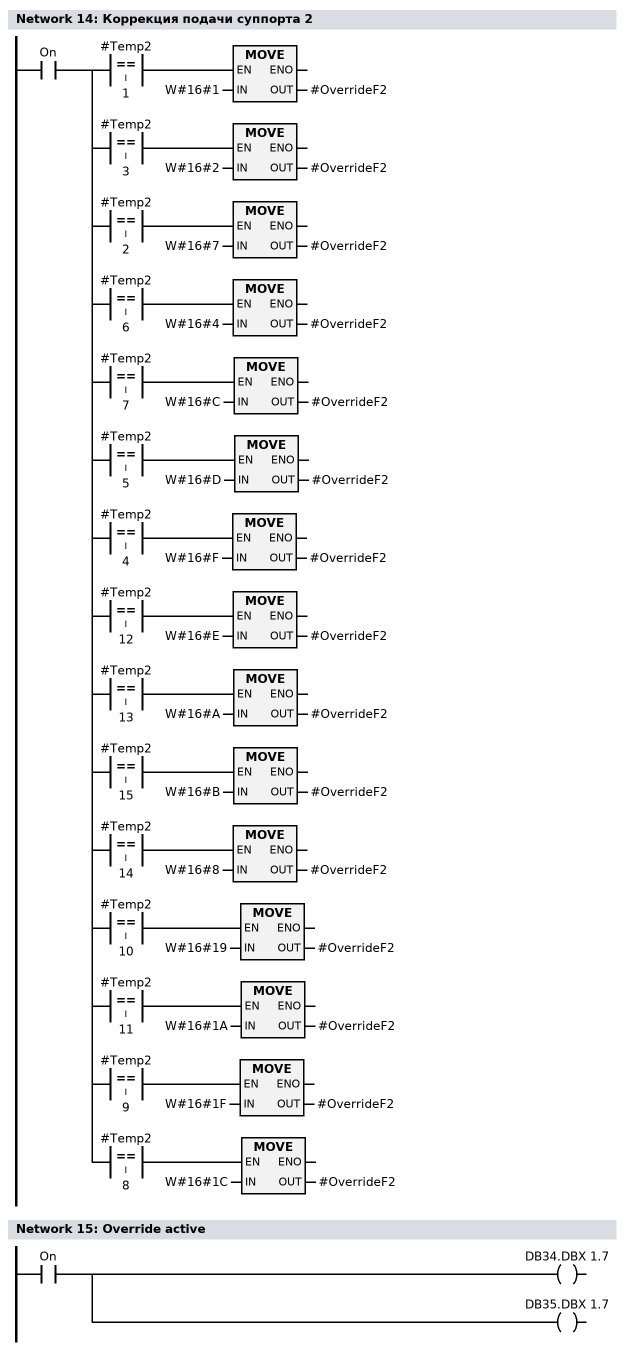
[picture p48: Correction networks 14-15]
NETWORK
TITLE = Коррекция подачи суппорта 2
      A     "On";
      =     L 19.0;
      A     L 19.0;
      A(;
      L     #Temp2;
      L     1;
      ==I;
      );
      JNB   _01b;
      L     W#16#1;
      T     #OverrideF2;
_01b: NOP   0;
      A     L 19.0;
      A(;
      L     #Temp2;
      L     3;
      ==I;
      );
      JNB   _01c;
      L     W#16#2;
      T     #OverrideF2;
_01c: NOP   0;
      A     L 19.0;
      A(;
      L     #Temp2;
      L     2;
      ==I;
      );
      JNB   _01d;
      L     W#16#7;
      T     #OverrideF2;
_01d: NOP   0;
      A     L 19.0;
      A(;
      L     #Temp2;
      L     6;
      ==I;
      );
      JNB   _01e;
      L     W#16#4;
      T     #OverrideF2;
_01e: NOP   0;
      A     L 19.0;
      A(;
      L     #Temp2;
      L     7;
      ==I;
      );
      JNB   _01f;
      L     W#16#C;
      T     #OverrideF2;
_01f: NOP   0;
      A     L 19.0;
      A(;
      L     #Temp2;
      L     5;
      ==I;
      );
      JNB   _020;
      L     W#16#D;
      T     #OverrideF2;
_020: NOP   0;
      A     L 19.0;
      A(;
      L     #Temp2;
      L     4;
      ==I;
      );
      JNB   _021;
      L     W#16#F;
      T     #OverrideF2;
_021: NOP   0;
      A     L 19.0;
      A(;
      L     #Temp2;
      L     12;
      ==I;
      );
      JNB   _022;
      L     W#16#E;
      T     #OverrideF2;
_022: NOP   0;
      A     L 19.0;
      A(;
      L     #Temp2;
      L     13;
      ==I;
      );
      JNB   _023;
      L     W#16#A;
      T     #OverrideF2;
_023: NOP   0;
      A     L 19.0;
      A(;
      L     #Temp2;
      L     15;
      ==I;
      );
      JNB   _024;
      L     W#16#B;
      T     #OverrideF2;
_024: NOP   0;
      A     L 19.0;
      A(;
      L     #Temp2;
      L     14;
      ==I;
      );
      JNB   _025;
      L     W#16#8;
      T     #OverrideF2;
_025: NOP   0;
      A     L 19.0;
      A(;
      L     #Temp2;
      L     10;
      ==I;
      );
      JNB   _026;
      L     W#16#19;
      T     #OverrideF2;
_026: NOP   0;
      A     L 19.0;
      A(;
      L     #Temp2;
      L     11;
      ==I;
      );
      JNB   _027;
      L     W#16#1A;
      T     #OverrideF2;
_027: NOP   0;
      A     L 19.0;
      A(;
      L     #Temp2;
      L     9;
      ==I;
      );
      JNB   _028;
      L     W#16#1F;
      T     #OverrideF2;
_028: NOP   0;
      A     L 19.0;
      A(;
      L     #Temp2;
      L     8;
      ==I;
      );
      JNB   _029;
      L     W#16#1C;
      T     #OverrideF2;
_029: NOP   0;
NETWORK
TITLE = Override active
      A     "On";
      =     DB34.DBX 1.7;
      =     DB35.DBX 1.7;
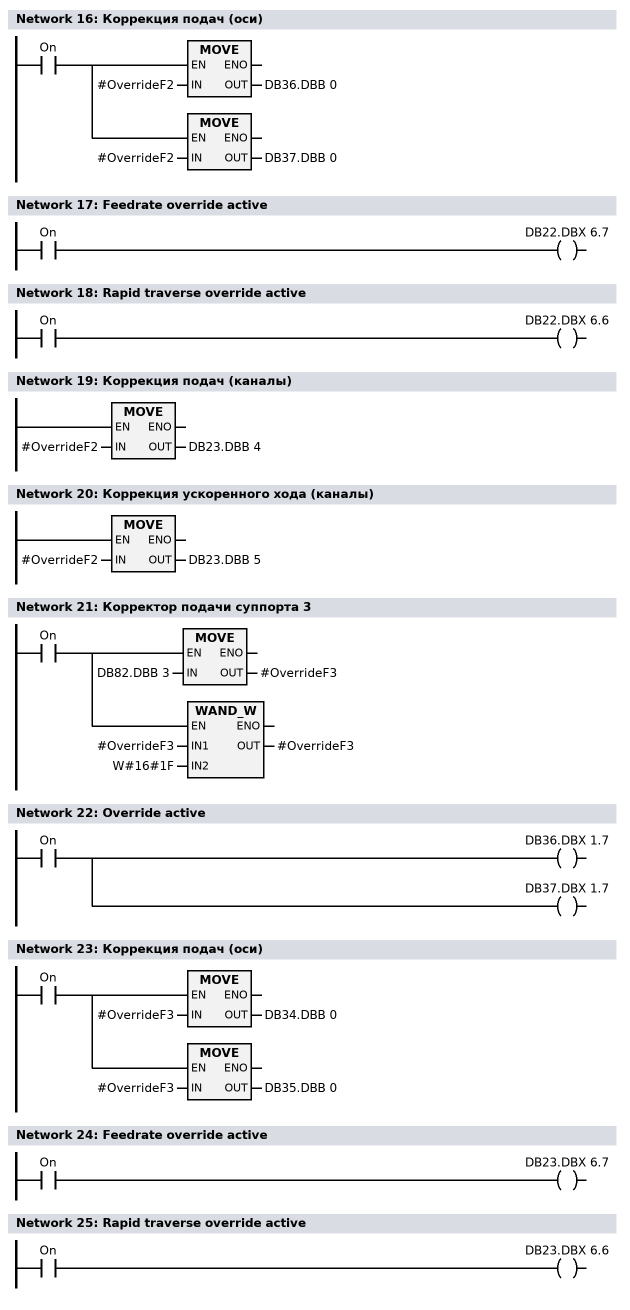
NETWORK
TITLE = Коррекция подач (оси)
      A     "On";
      =     L 19.0;
      A     L 19.0;
      JNB   _02a;
      L     #OverrideF2;
      T     DB36.DBB 0;
_02a: NOP   0;
      A     L 19.0;
      JNB   _02b;
      L     #OverrideF2;
      T     DB37.DBB 0;
_02b: NOP   0;
NETWORK
TITLE = Feedrate override active
      A     "On";
      =     DB22.DBX 6.7;
NETWORK
TITLE = Rapid traverse override active
      A     "On";
      =     DB22.DBX 6.6;
NETWORK
TITLE = Коррекция подач (каналы)
      L     #OverrideF2;
      T     DB23.DBB 4;
      NOP   0;
NETWORK
TITLE = Коррекция ускоренного хода (каналы)
      L     #OverrideF2;
      T     DB23.DBB 5;
      NOP   0;
NETWORK
TITLE = Корректор подачи суппорта 3
      A     "On";
      =     L 19.0;
      A     L 19.0;
      JNB   _02c;
      L     DB82.DBB 3;
      T     #OverrideF3;
_02c: NOP   0;
      A     L 19.0;
      JNB   _02d;
      L     #OverrideF3;
      L     W#16#1F;
      AW;
      T     #OverrideF3;
_02d: NOP   0;
NETWORK
TITLE = Override active
      A     "On";
      =     DB36.DBX 1.7;
      =     DB37.DBX 1.7;
NETWORK
TITLE = Коррекция подач (оси)
      A     "On";
      =     L 19.0;
      A     L 19.0;
      JNB   _02e;
      L     #OverrideF3;
      T     DB34.DBB 0;
_02e: NOP   0;
      A     L 19.0;
      JNB   _02f;
      L     #OverrideF3;
      T     DB35.DBB 0;
_02f: NOP   0;
NETWORK
TITLE = Feedrate override active
      A     "On";
      =     DB23.DBX 6.7;
NETWORK
TITLE = Rapid traverse override active
      A     "On";
      =     DB23.DBX 6.6;
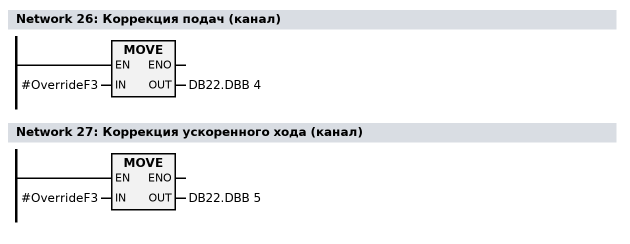
NETWORK
TITLE = Коррекция подач (канал)
      L     #OverrideF3;
      T     DB22.DBB 4;
      NOP   0;
NETWORK
TITLE = Коррекция ускоренного хода (канал)
      L     #OverrideF3;
      T     DB22.DBB 5;
      NOP   0;
NETWORK
TITLE = Корректор подачи суппорта 4
      A     "On";
      =     L 19.0;
      A     L 19.0;
      JNB   _030;
      L     DB82.DBB 0;
      T     #Temp1;
_030: NOP   0;
      A     L 19.0;
      JNB   _031;
      L     #Temp1;
      L     W#16#F0;
      AW;
      T     #Temp1;
_031: NOP   0;
      A     L 19.0;
      JNB   _032;
      L     W#16#4;
      L     #Temp1;
      SRW;
      T     #Temp1;
_032: NOP   0;
      A     L 19.0;
      JNB   _033;
      L     #Temp1;
      T     #Temp2;
_033: NOP   0;
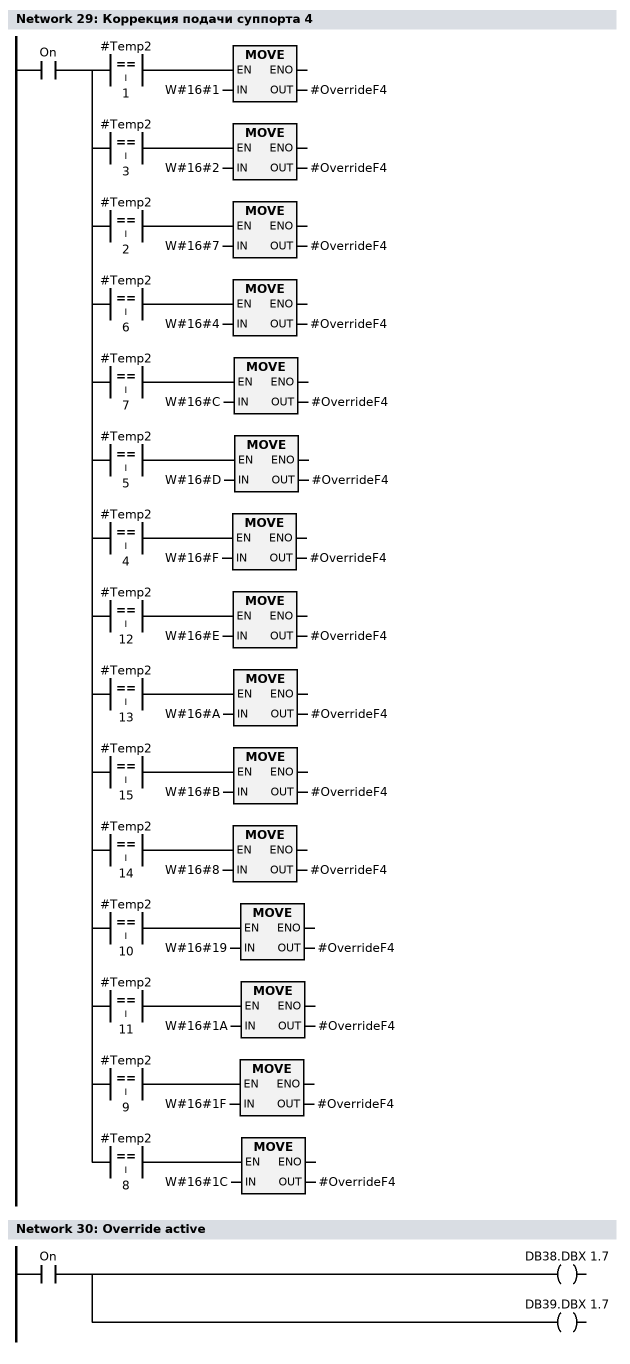
NETWORK
TITLE = Коррекция подачи суппорта 4
      A     "On";
      =     L 19.0;
      A     L 19.0;
      A(;
      L     #Temp2;
      L     1;
      ==I;
      );
      JNB   _034;
      L     W#16#1;
      T     #OverrideF4;
_034: NOP   0;
      A     L 19.0;
      A(;
      L     #Temp2;
      L     3;
      ==I;
      );
      JNB   _035;
      L     W#16#2;
      T     #OverrideF4;
_035: NOP   0;
      A     L 19.0;
      A(;
      L     #Temp2;
      L     2;
      ==I;
      );
      JNB   _036;
      L     W#16#7;
      T     #OverrideF4;
_036: NOP   0;
      A     L 19.0;
      A(;
      L     #Temp2;
      L     6;
      ==I;
      );
      JNB   _037;
      L     W#16#4;
      T     #OverrideF4;
_037: NOP   0;
      A     L 19.0;
      A(;
      L     #Temp2;
      L     7;
      ==I;
      );
      JNB   _038;
      L     W#16#C;
      T     #OverrideF4;
_038: NOP   0;
      A     L 19.0;
      A(;
      L     #Temp2;
      L     5;
      ==I;
      );
      JNB   _039;
      L     W#16#D;
      T     #OverrideF4;
_039: NOP   0;
      A     L 19.0;
      A(;
      L     #Temp2;
      L     4;
      ==I;
      );
      JNB   _03a;
      L     W#16#F;
      T     #OverrideF4;
_03a: NOP   0;
      A     L 19.0;
      A(;
      L     #Temp2;
      L     12;
      ==I;
      );
      JNB   _03b;
      L     W#16#E;
      T     #OverrideF4;
_03b: NOP   0;
      A     L 19.0;
      A(;
      L     #Temp2;
      L     13;
      ==I;
      );
      JNB   _03c;
      L     W#16#A;
      T     #OverrideF4;
_03c: NOP   0;
      A     L 19.0;
      A(;
      L     #Temp2;
      L     15;
      ==I;
      );
      JNB   _03d;
      L     W#16#B;
      T     #OverrideF4;
_03d: NOP   0;
      A     L 19.0;
      A(;
      L     #Temp2;
      L     14;
      ==I;
      );
      JNB   _03e;
      L     W#16#8;
      T     #OverrideF4;
_03e: NOP   0;
      A     L 19.0;
      A(;
      L     #Temp2;
      L     10;
      ==I;
      );
      JNB   _03f;
      L     W#16#19;
      T     #OverrideF4;
_03f: NOP   0;
      A     L 19.0;
      A(;
      L     #Temp2;
      L     11;
      ==I;
      );
      JNB   _040;
      L     W#16#1A;
      T     #OverrideF4;
_040: NOP   0;
      A     L 19.0;
      A(;
      L     #Temp2;
      L     9;
      ==I;
      );
      JNB   _041;
      L     W#16#1F;
      T     #OverrideF4;
_041: NOP   0;
      A     L 19.0;
      A(;
      L     #Temp2;
      L     8;
      ==I;
      );
      JNB   _042;
      L     W#16#1C;
      T     #OverrideF4;
_042: NOP   0;
NETWORK
TITLE = Override active
      A     "On";
      =     DB38.DBX 1.7;
      =     DB39.DBX 1.7;
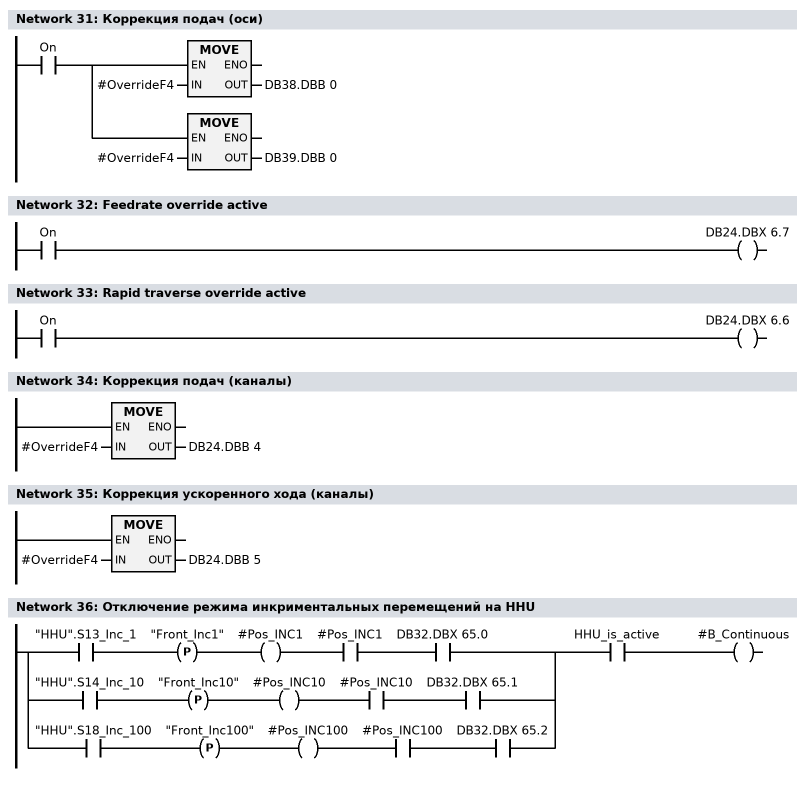
NETWORK
TITLE = Коррекция подач (оси)
      A     "On";
      =     L 19.0;
      A     L 19.0;
      JNB   _043;
      L     #OverrideF4;
      T     DB38.DBB 0;
_043: NOP   0;
      A     L 19.0;
      JNB   _044;
      L     #OverrideF4;
      T     DB39.DBB 0;
_044: NOP   0;
NETWORK
TITLE = Feedrate override active
      A     "On";
      =     DB24.DBX 6.7;
NETWORK
TITLE = Rapid traverse override active
      A     "On";
      =     DB24.DBX 6.6;
NETWORK
TITLE = Коррекция подач (каналы)
      L     #OverrideF4;
      T     DB24.DBB 4;
      NOP   0;
NETWORK
TITLE = Коррекция ускоренного хода (каналы)
      L     #OverrideF4;
      T     DB24.DBB 5;
      NOP   0;
NETWORK
TITLE = Отключение режима инкриментальных перемещений на HHU
      A(;
      A(;
      A     "HHU".S13_Inc_1;
      BLD   100;
      FP    "Front_Inc1";
      );
      =     #Pos_INC1;
      A     #Pos_INC1;
      A     DB32.DBX 65.0;
      O(;
      A(;
      A     "HHU".S14_Inc_10;
      BLD   100;
      FP    "Front_Inc10";
      );
      =     #Pos_INC10;
      A     #Pos_INC10;
      A     DB32.DBX 65.1;
      );
      O(;
      A(;
      A     "HHU".S18_Inc_100;
      BLD   100;
      FP    "Front_Inc100";
      );
      =     #Pos_INC100;
      A     #Pos_INC100;
      A     DB32.DBX 65.2;
      );
      );
      A     "HHU_is_active";
      =     #B_Continuous;
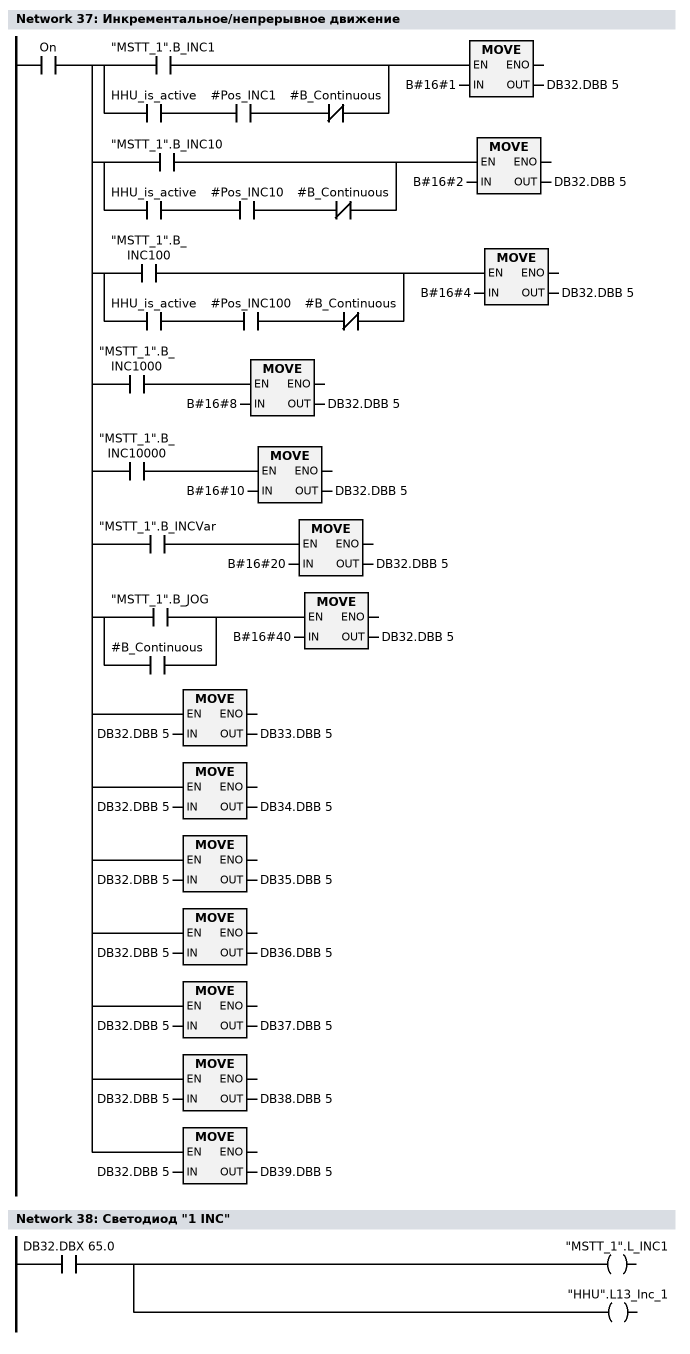
NETWORK
TITLE = Инкрементальное/непрерывное движение
      A     "On";
      =     L 19.0;
      A     L 19.0;
      A(;
      O     "MSTT_1".B_INC1;
      O;
      A     "HHU_is_active";
      A     #Pos_INC1;
      AN    #B_Continuous;
      );
      JNB   _045;
      L     B#16#1;
      T     DB32.DBB 5;
_045: NOP   0;
      A     L 19.0;
      A(;
      O     "MSTT_1".B_INC10;
      O;
      A     "HHU_is_active";
      A     #Pos_INC10;
      AN    #B_Continuous;
      );
      JNB   _046;
      L     B#16#2;
      T     DB32.DBB 5;
_046: NOP   0;
      A     L 19.0;
      A(;
      O     "MSTT_1".B_INC100;
      O;
      A     "HHU_is_active";
      A     #Pos_INC100;
      AN    #B_Continuous;
      );
      JNB   _047;
      L     B#16#4;
      T     DB32.DBB 5;
_047: NOP   0;
      A     L 19.0;
      A     "MSTT_1".B_INC1000;
      JNB   _048;
      L     B#16#8;
      T     DB32.DBB 5;
_048: NOP   0;
      A     L 19.0;
      A     "MSTT_1".B_INC10000;
      JNB   _049;
      L     B#16#10;
      T     DB32.DBB 5;
_049: NOP   0;
      A     L 19.0;
      A     "MSTT_1".B_INCVar;
      JNB   _04a;
      L     B#16#20;
      T     DB32.DBB 5;
_04a: NOP   0;
      A     L 19.0;
      A(;
      O     "MSTT_1".B_JOG;
      O     #B_Continuous;
      );
      JNB   _04b;
      L     B#16#40;
      T     DB32.DBB 5;
_04b: NOP   0;
      A     L 19.0;
      JNB   _04c;
      L     DB32.DBB 5;
      T     DB33.DBB 5;
_04c: NOP   0;
      A     L 19.0;
      JNB   _04d;
      L     DB32.DBB 5;
      T     DB34.DBB 5;
_04d: NOP   0;
      A     L 19.0;
      JNB   _04e;
      L     DB32.DBB 5;
      T     DB35.DBB 5;
_04e: NOP   0;
      A     L 19.0;
      JNB   _04f;
      L     DB32.DBB 5;
      T     DB36.DBB 5;
_04f: NOP   0;
      A     L 19.0;
      JNB   _050;
      L     DB32.DBB 5;
      T     DB37.DBB 5;
_050: NOP   0;
      A     L 19.0;
      JNB   _051;
      L     DB32.DBB 5;
      T     DB38.DBB 5;
_051: NOP   0;
      A     L 19.0;
      JNB   _052;
      L     DB32.DBB 5;
      T     DB39.DBB 5;
_052: NOP   0;
NETWORK
TITLE = Светодиод "1 INC"
      A     DB32.DBX 65.0;
      =     "MSTT_1".L_INC1;
      =     "HHU".L13_Inc_1;
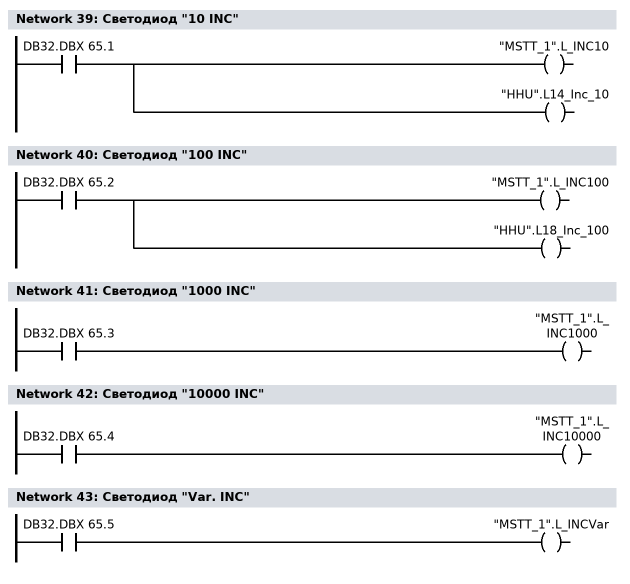
NETWORK
TITLE = Светодиод "10 INC"
      A     DB32.DBX 65.1;
      =     "MSTT_1".L_INC10;
      =     "HHU".L14_Inc_10;
NETWORK
TITLE = Светодиод "100 INC"
      A     DB32.DBX 65.2;
      =     "MSTT_1".L_INC100;
      =     "HHU".L18_Inc_100;
NETWORK
TITLE = Светодиод "1000 INC"
      A     DB32.DBX 65.3;
      =     "MSTT_1".L_INC1000;
NETWORK
TITLE = Светодиод "10000 INC"
      A     DB32.DBX 65.4;
      =     "MSTT_1".L_INC10000;
NETWORK
TITLE = Светодиод "Var. INC"
      A     DB32.DBX 65.5;
      =     "MSTT_1".L_INCVar;
END_FUNCTION

FUNCTION "Others" : VOID	// FC 112
AUTHOR : SEDIN
VERSION : 0.1
VAR_TEMP
  F_Ret_Val : INT ;
  Alarms1 : DINT ;
END_VAR
BEGIN
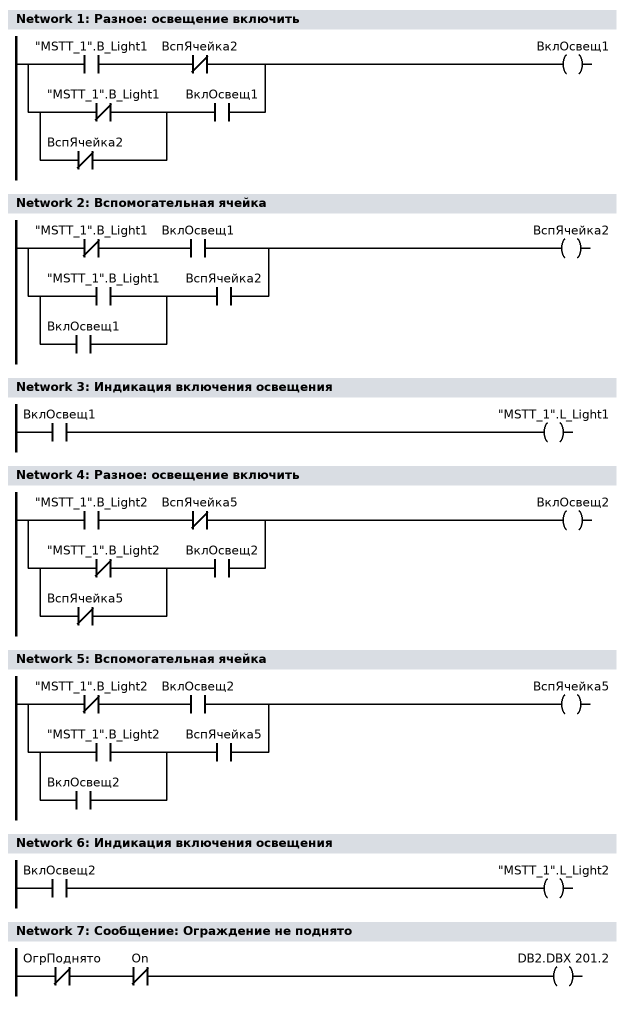
NETWORK
TITLE = Разное: освещение включить
      A     "MSTT_1".B_Light1;
      AN    "ВспЯчейка2";
      O;
      A(;
      ON    "MSTT_1".B_Light1;
      ON    "ВспЯчейка2";
      );
      A     "ВклОсвещ1";
      =     "ВклОсвещ1";
NETWORK
TITLE = Вспомогательная ячейка
      AN    "MSTT_1".B_Light1;
      A     "ВклОсвещ1";
      O;
      A(;
      O     "MSTT_1".B_Light1;
      O     "ВклОсвещ1";
      );
      A     "ВспЯчейка2";
      =     "ВспЯчейка2";
NETWORK
TITLE = Индикация включения освещения
      A     "ВклОсвещ1";
      =     "MSTT_1".L_Light1;
NETWORK
TITLE = Разное: освещение включить
      A     "MSTT_1".B_Light2;
      AN    "ВспЯчейка5";
      O;
      A(;
      ON    "MSTT_1".B_Light2;
      ON    "ВспЯчейка5";
      );
      A     "ВклОсвещ2";
      =     "ВклОсвещ2";
NETWORK
TITLE = Вспомогательная ячейка
      AN    "MSTT_1".B_Light2;
      A     "ВклОсвещ2";
      O;
      A(;
      O     "MSTT_1".B_Light2;
      O     "ВклОсвещ2";
      );
      A     "ВспЯчейка5";
      =     "ВспЯчейка5";
NETWORK
TITLE = Индикация включения освещения
      A     "ВклОсвещ2";
      =     "MSTT_1".L_Light2;
NETWORK
TITLE = Сообщение: Ограждение не поднято
      AN    "ОгрПоднято";
      AN    "On";
      =     DB2.DBX 201.2;
END_FUNCTION

FUNCTION "Hydraullics" : VOID	// FC 115
AUTHOR : SEDIN
VERSION : 0.1
BEGIN
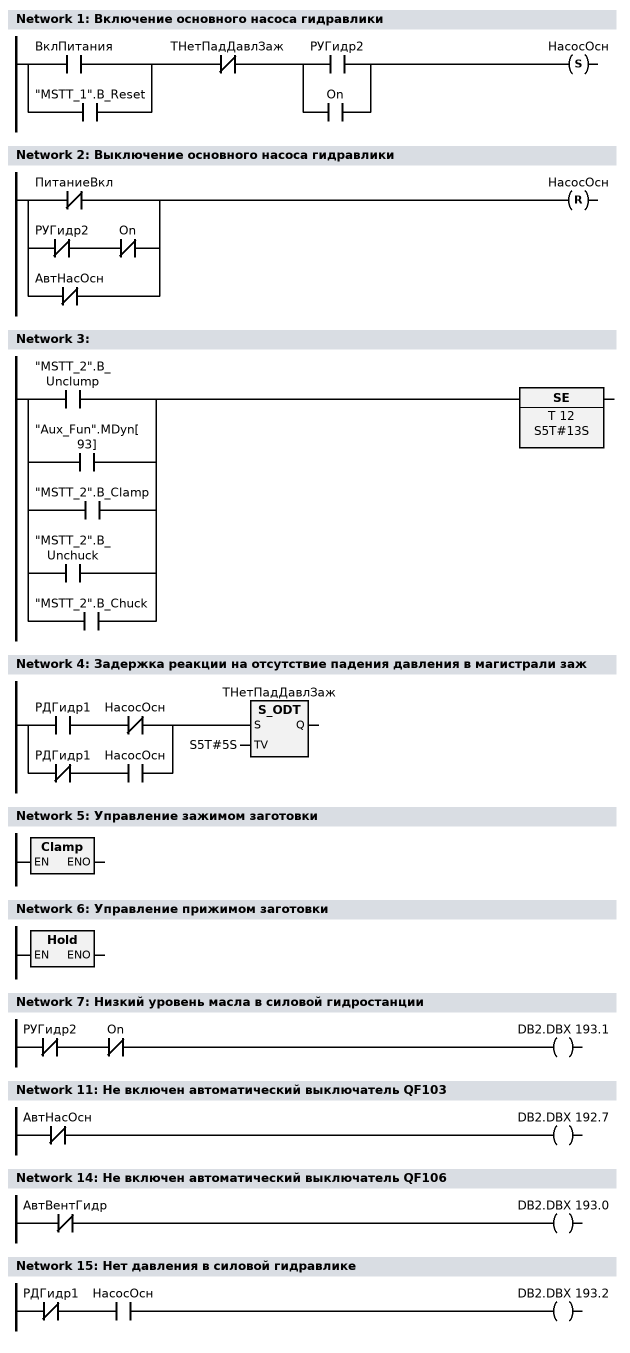
NETWORK
TITLE = Включение основного насоса гидравлики
      A(;
      O     "ВклПитания";
      O     "MSTT_1".B_Reset;
      );
      AN    "ТНетПадДавлЗаж";
      A(;
      O     "РУГидр2";
      O     "On";
      );
      S     "НасосОсн";
NETWORK
TITLE = Выключение основного насоса гидравлики
      ON    "ПитаниеВкл";
      O;
      AN    "РУГидр2";
      AN    "On";
      ON    "АвтНасОсн";
      R     "НасосОсн";
NETWORK
TITLE =
      O     "MSTT_2".B_Unclump;
      O     "Aux_Fun".MDyn[93];
      O     "MSTT_2".B_Clamp;
      O     "MSTT_2".B_Unchuck;
      O     "MSTT_2".B_Chuck;
      L     S5T#13S;
      SE    T 12;
NETWORK
TITLE = Задержка реакции на отсутствие падения давления в магистрали заж
      A(;
      A     "РДГидр1";
      AN    "НасосОсн";
      O;
      AN    "РДГидр1";
      A     "НасосОсн";
      );
      L     S5T#5S;
      SD    "ТНетПадДавлЗаж";
      NOP   0;
      NOP   0;
      NOP   0;
      NOP   0;
NETWORK
TITLE = Управление зажимом заготовки
      CALL  "Clamp";
      NOP   0;
NETWORK
TITLE = Управление прижимом заготовки
      CALL  "Hold";
      NOP   0;
NETWORK
TITLE = Низкий уровень масла в силовой гидростанции
      AN    "РУГидр2";
      AN    "On";
      =     DB2.DBX 193.1;
NETWORK
TITLE = Фильтр SF101 в системе гидравлики засорен
//      AN    "ФильтрSF101"
//      AN    "On"
//      =     "ALMSG_DB".A7001xx[51]
NETWORK
TITLE = Фильтр SF102 в системе гидравлики засорен
//      AN    "ФильтрSF102"
//      AN    "On"
//      =     "ALMSG_DB".A7001xx[52]
NETWORK
TITLE = Фильтр SF103 в системе гидравлики засорен
//      AN    "ФильтрSF103"
//      AN    "On"
//      =     "ALMSG_DB".A7001xx[54]
NETWORK
TITLE = Не включен автоматический выключатель QF103
      AN    "АвтНасОсн";
      =     DB2.DBX 192.7;
NETWORK
TITLE = Не включен автоматический выключатель QF104
//      AN    "АвтНасПод"
//      AN    "On"
//      =     "ALMSG_DB".A7001xx[57]
NETWORK
TITLE = Не включен насос системы гидравлики
//      AN    "НасосОсн"
//      A     "ПитаниеВкл"
//      =     "ALMSG_DB".A7001xx[58]
NETWORK
TITLE = Не включен автоматический выключатель QF106
      AN    "АвтВентГидр";
      =     DB2.DBX 193.0;
NETWORK
TITLE = Нет давления в силовой гидравлике
      AN    "РДГидр1";
      A     "НасосОсн";
      =     DB2.DBX 193.2;
END_FUNCTION

FUNCTION "Clamp" : VOID	// FC 116
AUTHOR : SEDIN
VERSION : 0.1
BEGIN
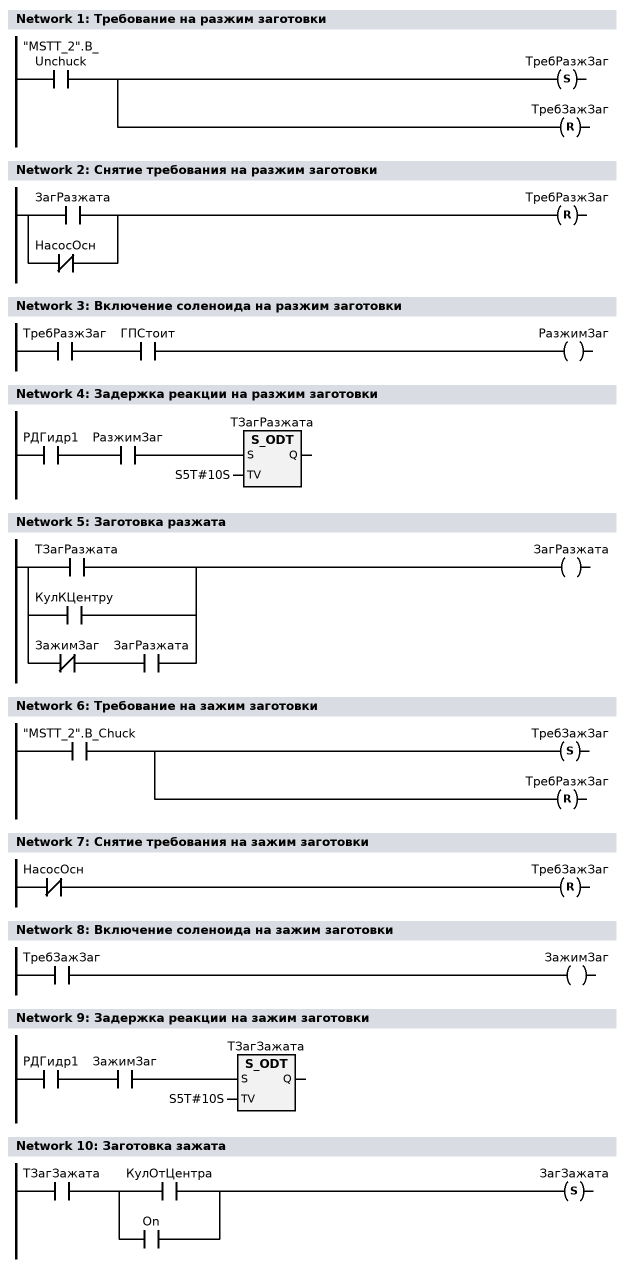
NETWORK
TITLE = Требование на разжим заготовки
      A     "MSTT_2".B_Unchuck;
      S     "ТребРазжЗаг";
      R     "ТребЗажЗаг";
NETWORK
TITLE = Снятие требования на разжим заготовки
      O     "ЗагРазжата";
      ON    "НасосОсн";
      R     "ТребРазжЗаг";
NETWORK
TITLE = Включение соленоида на разжим заготовки
      A     "ТребРазжЗаг";
      A     "ГПСтоит";
      =     "РазжимЗаг";
NETWORK
TITLE = Задержка реакции на разжим заготовки
      A     "РДГидр1";
      A     "РазжимЗаг";
      L     S5T#10S;
      SD    "ТЗагРазжата";
      NOP   0;
      NOP   0;
      NOP   0;
      NOP   0;
NETWORK
TITLE = Заготовка разжата
      O     "ТЗагРазжата";
      O     "КулКЦентру";
      O;
      AN    "ЗажимЗаг";
      A     "ЗагРазжата";
      =     "ЗагРазжата";
NETWORK
TITLE = Требование на зажим заготовки
      A     "MSTT_2".B_Chuck;
      S     "ТребЗажЗаг";
      R     "ТребРазжЗаг";
NETWORK
TITLE = Снятие требования на зажим заготовки
      AN    "НасосОсн";
      R     "ТребЗажЗаг";
NETWORK
TITLE = Включение соленоида на зажим заготовки
      A     "ТребЗажЗаг";
      =     "ЗажимЗаг";
NETWORK
TITLE = Задержка реакции на зажим заготовки
      A     "РДГидр1";
      A     "ЗажимЗаг";
      L     S5T#10S;
      SD    "ТЗагЗажата";
      NOP   0;
      NOP   0;
      NOP   0;
      NOP   0;
NETWORK
TITLE = Заготовка зажата
      A     "ТЗагЗажата";
      A(;
      O     "КулОтЦентра";
      O     "On";
      );
      S     "ЗагЗажата";
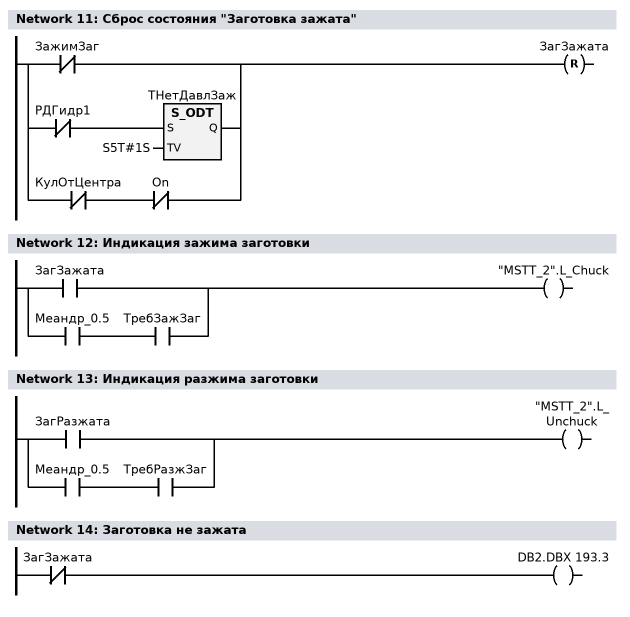
NETWORK
TITLE = Сброс состояния "Заготовка зажата"
      ON    "ЗажимЗаг";
      O(;
      AN    "РДГидр1";
      L     S5T#1S;
      SD    "ТНетДавлЗаж";
      NOP   0;
      NOP   0;
      NOP   0;
      A     "ТНетДавлЗаж";
      );
      O;
      AN    "КулОтЦентра";
      AN    "On";
      R     "ЗагЗажата";
NETWORK
TITLE = Индикация зажима заготовки
      O     "ЗагЗажата";
      O;
      A     "Меандр_0.5";
      A     "ТребЗажЗаг";
      =     "MSTT_2".L_Chuck;
NETWORK
TITLE = Индикация разжима заготовки
      O     "ЗагРазжата";
      O;
      A     "Меандр_0.5";
      A     "ТребРазжЗаг";
      =     "MSTT_2".L_Unchuck;
NETWORK
TITLE = Заготовка не зажата
      AN    "ЗагЗажата";
      =     DB2.DBX 193.3;
END_FUNCTION

FUNCTION "Hold" : VOID	// FC 118
AUTHOR : SEDIN
VERSION : 0.1
BEGIN
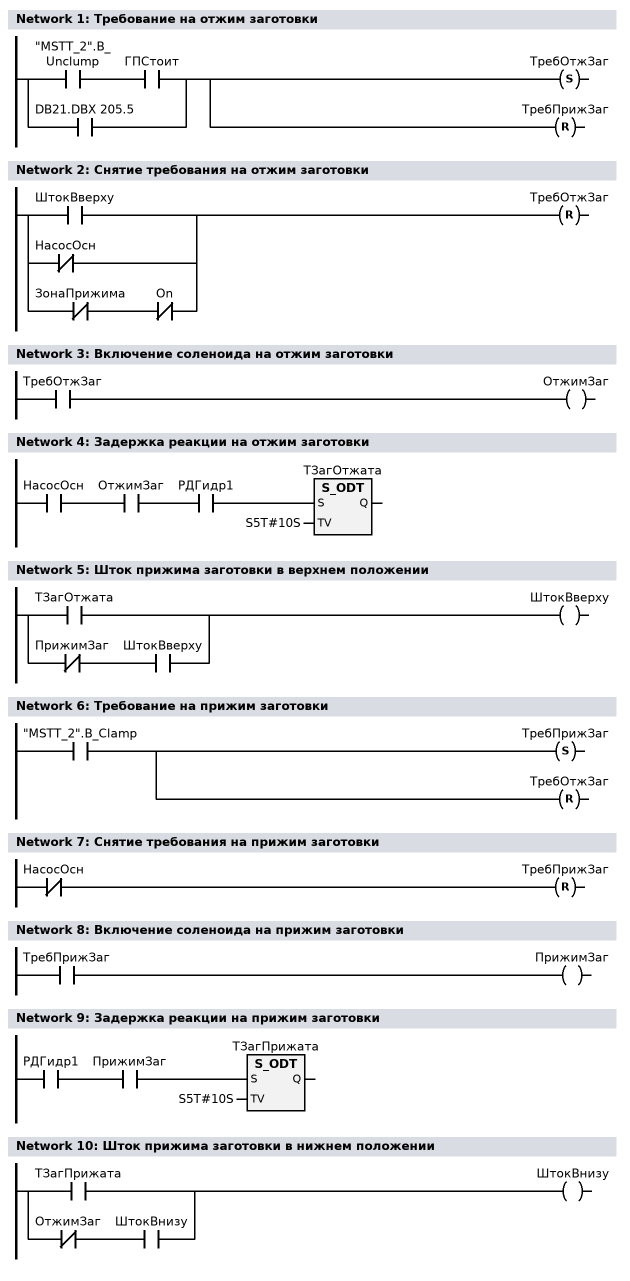
NETWORK
TITLE = Требование на отжим заготовки
      A     "MSTT_2".B_Unclump;
      A     "ГПСтоит";
      O     DB21.DBX 205.5;
      S     "ТребОтжЗаг";
      R     "ТребПрижЗаг";
NETWORK
TITLE = Снятие требования на отжим заготовки
      O     "ШтокВверху";
      ON    "НасосОсн";
      O;
      AN    "ЗонаПрижима";
      AN    "On";
      R     "ТребОтжЗаг";
NETWORK
TITLE = Включение соленоида на отжим заготовки
      A     "ТребОтжЗаг";
      =     "ОтжимЗаг";
NETWORK
TITLE = Задержка реакции на отжим заготовки
      A     "НасосОсн";
      A     "ОтжимЗаг";
      A     "РДГидр1";
      L     S5T#10S;
      SD    "ТЗагОтжата";
      NOP   0;
      NOP   0;
      NOP   0;
      NOP   0;
NETWORK
TITLE = Шток прижима заготовки в верхнем положении
      O     "ТЗагОтжата";
      O;
      AN    "ПрижимЗаг";
      A     "ШтокВверху";
      =     "ШтокВверху";
NETWORK
TITLE = Требование на прижим заготовки
      A     "MSTT_2".B_Clamp;
      S     "ТребПрижЗаг";
      R     "ТребОтжЗаг";
NETWORK
TITLE = Снятие требования на прижим заготовки
      AN    "НасосОсн";
      R     "ТребПрижЗаг";
NETWORK
TITLE = Включение соленоида на прижим заготовки
      A     "ТребПрижЗаг";
      =     "ПрижимЗаг";
NETWORK
TITLE = Задержка реакции на прижим заготовки
      A     "РДГидр1";
      A     "ПрижимЗаг";
      L     S5T#10S;
      SD    "ТЗагПрижата";
      NOP   0;
      NOP   0;
      NOP   0;
      NOP   0;
NETWORK
TITLE = Шток прижима заготовки в нижнем положении
      O     "ТЗагПрижата";
      O;
      AN    "ОтжимЗаг";
      A     "ШтокВнизу";
      =     "ШтокВнизу";
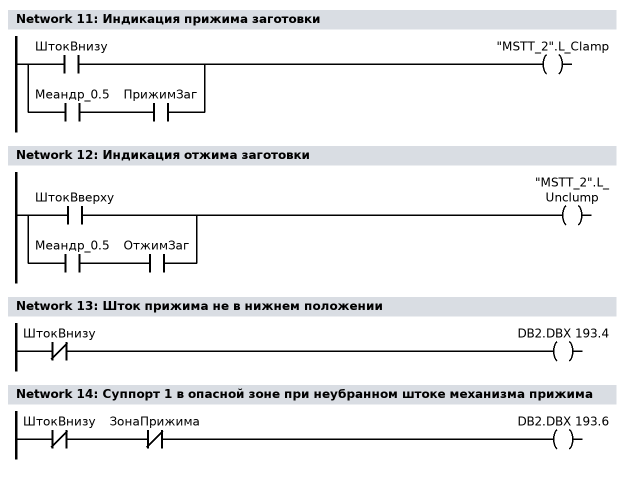
NETWORK
TITLE = Индикация прижима заготовки
      O     "ШтокВнизу";
      O;
      A     "Меандр_0.5";
      A     "ПрижимЗаг";
      =     "MSTT_2".L_Clamp;
NETWORK
TITLE = Индикация отжима заготовки
      O     "ШтокВверху";
      O;
      A     "Меандр_0.5";
      A     "ОтжимЗаг";
      =     "MSTT_2".L_Unclump;
NETWORK
TITLE = Шток прижима не в нижнем положении
      AN    "ШтокВнизу";
      =     DB2.DBX 193.4;
NETWORK
TITLE = Суппорт 1 в опасной зоне при неубранном штоке механизма прижима
      AN    "ШтокВнизу";
      AN    "ЗонаПрижима";
      =     DB2.DBX 193.6;
END_FUNCTION

FUNCTION "Table_Lub" : VOID	// FC 120
AUTHOR : SEDIN
VERSION : 0.1
BEGIN
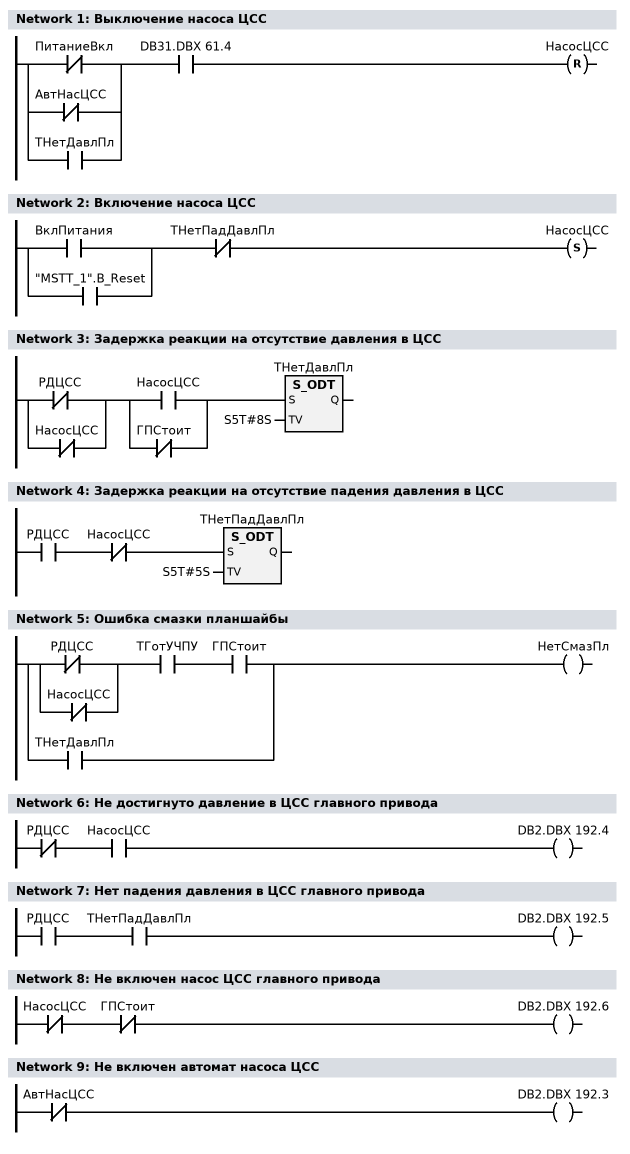
NETWORK
TITLE = Выключение насоса ЦСС
      A(;
      ON    "ПитаниеВкл";
      ON    "АвтНасЦСС";
      O     "ТНетДавлПл";
      );
      A     DB31.DBX 61.4;
      R     "НасосЦСС";
NETWORK
TITLE = Включение насоса ЦСС
      A(;
      O     "ВклПитания";
      O     "MSTT_1".B_Reset;
      );
      AN    "ТНетПадДавлПл";
      S     "НасосЦСС";
NETWORK
TITLE = Задержка реакции на отсутствие давления в ЦСС
      A(;
      ON    "РДЦСС";
      ON    "НасосЦСС";
      );
      A(;
      O     "НасосЦСС";
      ON    "ГПСтоит";
      );
      L     S5T#8S;
      SD    "ТНетДавлПл";
      NOP   0;
      NOP   0;
      NOP   0;
      NOP   0;
NETWORK
TITLE = Задержка реакции на отсутствие падения давления в ЦСС
      A     "РДЦСС";
      AN    "НасосЦСС";
      L     S5T#5S;
      SD    "ТНетПадДавлПл";
      NOP   0;
      NOP   0;
      NOP   0;
      NOP   0;
NETWORK
TITLE = Ошибка смазки планшайбы
      A(;
      ON    "РДЦСС";
      ON    "НасосЦСС";
      );
      A     "ТГотУЧПУ";
      A     "ГПСтоит";
      O     "ТНетДавлПл";
      =     "НетСмазПл";
NETWORK
TITLE = Не достигнуто давление в ЦСС главного привода
      AN    "РДЦСС";
      A     "НасосЦСС";
      =     DB2.DBX 192.4;
NETWORK
TITLE = Нет падения давления в ЦСС главного привода
      A     "РДЦСС";
      A     "ТНетПадДавлПл";
      =     DB2.DBX 192.5;
NETWORK
TITLE = Не включен насос ЦСС главного привода
      AN    "НасосЦСС";
      AN    "ГПСтоит";
      =     DB2.DBX 192.6;
NETWORK
TITLE = Не включен автомат насоса ЦСС
      AN    "АвтНасЦСС";
      =     DB2.DBX 192.3;
END_FUNCTION

FUNCTION "MiniHHU" : VOID	// FC 121
VERSION : 0.1
BEGIN
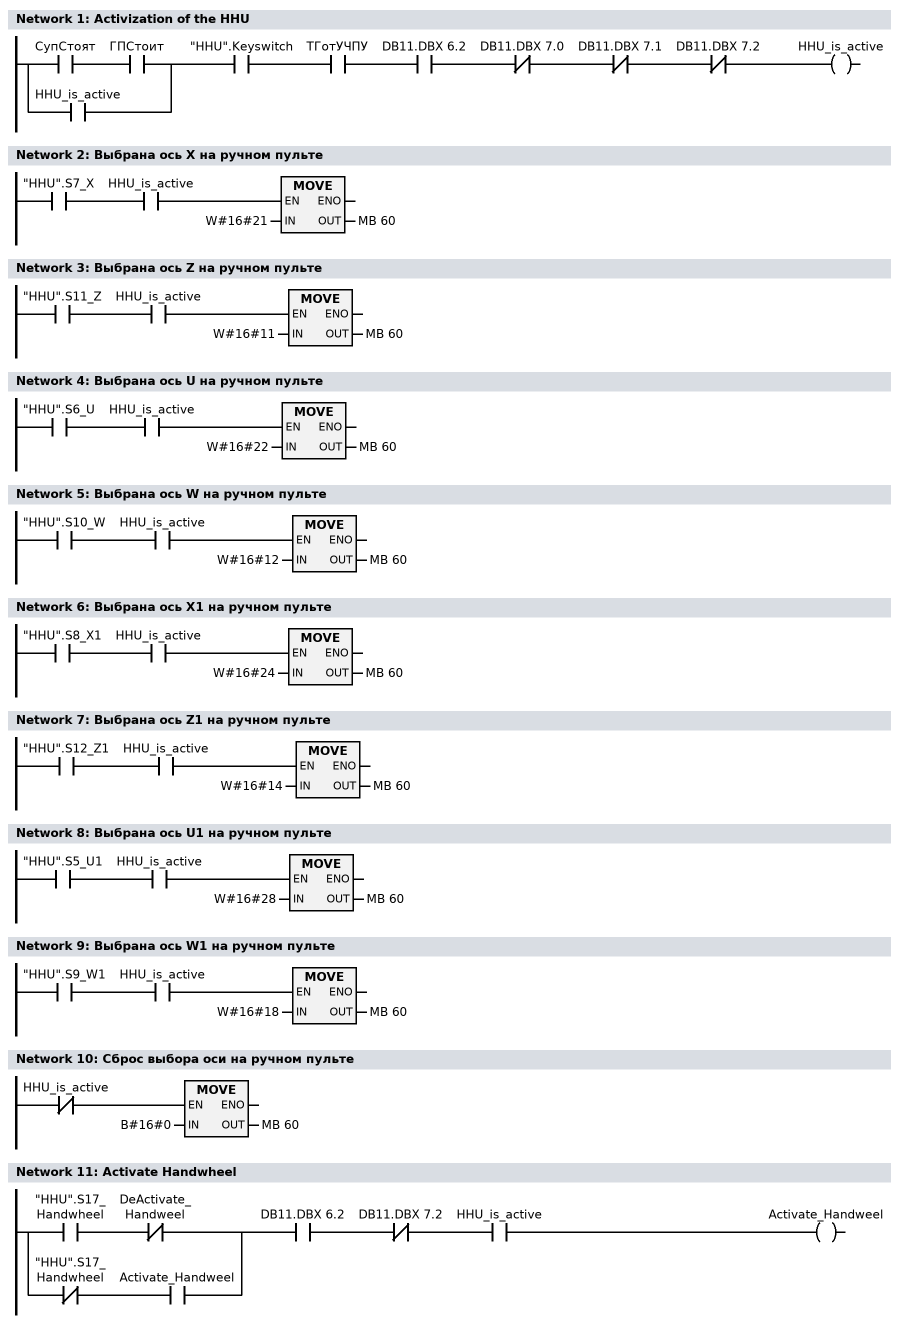
NETWORK
TITLE = Activization of the HHU
      A(;
      A     "СупСтоят";
      A     "ГПСтоит";
      O     "HHU_is_active";
      );
      A     "HHU".Keyswitch;
      A     "ТГотУЧПУ";
      A     DB11.DBX 6.2;
      AN    DB11.DBX 7.0;
      AN    DB11.DBX 7.1;
      AN    DB11.DBX 7.2;
      =     "HHU_is_active";
NETWORK
TITLE = Выбрана ось X на ручном пульте
      A     "HHU".S7_X;
      A     "HHU_is_active";
      JNB   _001;
      L     W#16#21;
      T     MB 60;
_001: NOP   0;
NETWORK
TITLE = Выбрана ось Z на ручном пульте
      A     "HHU".S11_Z;
      A     "HHU_is_active";
      JNB   _002;
      L     W#16#11;
      T     MB 60;
_002: NOP   0;
NETWORK
TITLE = Выбрана ось U на ручном пульте
      A     "HHU".S6_U;
      A     "HHU_is_active";
      JNB   _003;
      L     W#16#22;
      T     MB 60;
_003: NOP   0;
NETWORK
TITLE = Выбрана ось W на ручном пульте
      A     "HHU".S10_W;
      A     "HHU_is_active";
      JNB   _004;
      L     W#16#12;
      T     MB 60;
_004: NOP   0;
NETWORK
TITLE = Выбрана ось X1 на ручном пульте
      A     "HHU".S8_X1;
      A     "HHU_is_active";
      JNB   _005;
      L     W#16#24;
      T     MB 60;
_005: NOP   0;
NETWORK
TITLE = Выбрана ось Z1 на ручном пульте
      A     "HHU".S12_Z1;
      A     "HHU_is_active";
      JNB   _006;
      L     W#16#14;
      T     MB 60;
_006: NOP   0;
NETWORK
TITLE = Выбрана ось U1 на ручном пульте
      A     "HHU".S5_U1;
      A     "HHU_is_active";
      JNB   _007;
      L     W#16#28;
      T     MB 60;
_007: NOP   0;
NETWORK
TITLE = Выбрана ось W1 на ручном пульте
      A     "HHU".S9_W1;
      A     "HHU_is_active";
      JNB   _008;
      L     W#16#18;
      T     MB 60;
_008: NOP   0;
NETWORK
TITLE = Сброс выбора оси на ручном пульте
      AN    "HHU_is_active";
      JNB   _009;
      L     B#16#0;
      T     MB 60;
_009: NOP   0;
NETWORK
TITLE = Activate Handwheel
      A(;
      A     "HHU".S17_Handwheel;
      AN    "DeActivate_Handweel";
      O;
      AN    "HHU".S17_Handwheel;
      A     "Activate_Handweel";
      );
      A     DB11.DBX 6.2;
      AN    DB11.DBX 7.2;
      A     "HHU_is_active";
      =     "Activate_Handweel";
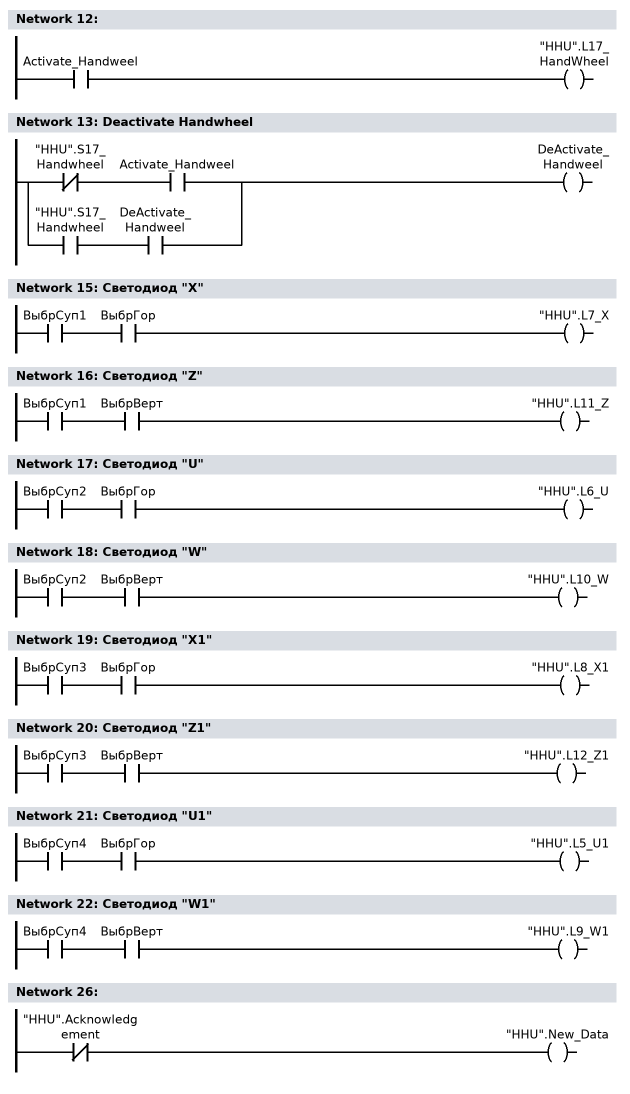
NETWORK
TITLE =
      A     "Activate_Handweel";
      =     "HHU".L17_HandWheel;
NETWORK
TITLE = Deactivate Handwheel
      AN    "HHU".S17_Handwheel;
      A     "Activate_Handweel";
      O;
      A     "HHU".S17_Handwheel;
      A     "DeActivate_Handweel";
      =     "DeActivate_Handweel";
NETWORK
TITLE =
NETWORK
TITLE = Светодиод "X"
      A     "ВыбрСуп1";
      A     "ВыбрГор";
      =     "HHU".L7_X;
NETWORK
TITLE = Светодиод "Z"
      A     "ВыбрСуп1";
      A     "ВыбрВерт";
      =     "HHU".L11_Z;
NETWORK
TITLE = Светодиод "U"
      A     "ВыбрСуп2";
      A     "ВыбрГор";
      =     "HHU".L6_U;
NETWORK
TITLE = Светодиод "W"
      A     "ВыбрСуп2";
      A     "ВыбрВерт";
      =     "HHU".L10_W;
NETWORK
TITLE = Светодиод "X1"
      A     "ВыбрСуп3";
      A     "ВыбрГор";
      =     "HHU".L8_X1;
NETWORK
TITLE = Светодиод "Z1"
      A     "ВыбрСуп3";
      A     "ВыбрВерт";
      =     "HHU".L12_Z1;
NETWORK
TITLE = Светодиод "U1"
      A     "ВыбрСуп4";
      A     "ВыбрГор";
      =     "HHU".L5_U1;
NETWORK
TITLE = Светодиод "W1"
      A     "ВыбрСуп4";
      A     "ВыбрВерт";
      =     "HHU".L9_W1;
NETWORK
TITLE =
      SET;
      S     DB83.DBX 6.7;
      A     "HHU".Acknowledgement;
      FP    "HHU".Auxilary[1];
      =     L 14.0;
      A     L 14.0;
      BLD   102;
      R     "HHU".New_Data;
      A     L 14.0;
      JNB   _010;
      L     DB83.DBB 7;
      INC   1;
      T     DB83.DBB 7;
_010: NOP   0;
      A     L 14.0;
      A     "HHU".Reserved_7_2;
      R     "HHU".Reserved_7_2;
NETWORK
TITLE =
      AN    "HHU".Keyswitch;
      =     L 15.0;
      A     L 15.0;
      AN    "HHU".Selection_Line_1_2;
      AN    "HHU".Selection_Line_3_4;
      JNB   _012;
      L     '$00';
      T     "HHU".DataLine[1];
      T     "HHU".DataLine[2];
      T     "HHU".DataLine[3];
      T     "HHU".DataLine[4];
      T     "HHU".DataLine[5];
      T     "HHU".DataLine[6];
      T     "HHU".DataLine[7];
      T     "HHU".DataLine[8];
      T     "HHU".DataLine[9];
      T     "HHU".DataLine[10];
      T     "HHU".DataLine[11];
      T     "HHU".DataLine[12];
      T     "HHU".DataLine[13];
      T     "HHU".DataLine[14];
      T     "HHU".DataLine[15];
      T     "HHU".DataLine[16];
_012: NOP   0;
      A     L 15.0;
      A     "HHU".Selection_Line_1_2;
      AN    "HHU".Selection_Line_3_4;
      JNB   _013;
      L     '$00';
      T     "HHU".DataLine[1];
      T     "HHU".DataLine[2];
      T     "HHU".DataLine[3];
      L     't';
      T     "HHU".DataLine[4];
      L     'o';
      T     "HHU".DataLine[5];
      L     'n';
      T     "HHU".DataLine[6];
      L     '$00';
      T     "HHU".DataLine[7];
      L     's';
      T     "HHU".DataLine[8];
      L     'i';
      T     "HHU".DataLine[9];
      L     '$00';
      T     "HHU".DataLine[10];
      L     '2';
      T     "HHU".DataLine[11];
      L     'T';
      T     "HHU".DataLine[12];
      L     'H';
      T     "HHU".DataLine[13];
      L     '$00';
      T     "HHU".DataLine[14];
      T     "HHU".DataLine[15];
      T     "HHU".DataLine[16];
_013: NOP   0;
      A     L 15.0;
      AN    "HHU".Selection_Line_1_2;
      A     "HHU".Selection_Line_3_4;
      JNB   _014;
      L     '$00';
      T     "HHU".DataLine[1];
      T     "HHU".DataLine[2];
      T     "HHU".DataLine[3];
      T     "HHU".DataLine[4];
      T     "HHU".DataLine[5];
      L     'e';
      T     "HHU".DataLine[6];
      L     'v';
      T     "HHU".DataLine[7];
      L     'i';
      T     "HHU".DataLine[8];
      L     't';
      T     "HHU".DataLine[9];
      L     'c';
      T     "HHU".DataLine[10];
      L     'a';
      T     "HHU".DataLine[11];
      L     '$00';
      T     "HHU".DataLine[12];
      T     "HHU".DataLine[13];
      T     "HHU".DataLine[14];
      T     "HHU".DataLine[15];
      T     "HHU".DataLine[16];
_014: NOP   0;
      A     L 15.0;
      A     "HHU".Selection_Line_1_2;
      A     "HHU".Selection_Line_3_4;
      JNB   _015;
      L     '$00';
      T     "HHU".DataLine[1];
      T     "HHU".DataLine[2];
      T     "HHU".DataLine[3];
      T     "HHU".DataLine[4];
      T     "HHU".DataLine[5];
      T     "HHU".DataLine[6];
      T     "HHU".DataLine[7];
      T     "HHU".DataLine[8];
      T     "HHU".DataLine[9];
      T     "HHU".DataLine[10];
      T     "HHU".DataLine[11];
      T     "HHU".DataLine[12];
      T     "HHU".DataLine[13];
      T     "HHU".DataLine[14];
      T     "HHU".DataLine[15];
      T     "HHU".DataLine[16];
_015: NOP   0;
NETWORK
TITLE =
      A     "HHU".Keyswitch;
      =     L 15.0;
      A     L 15.0;
      AN    "HHU".Selection_Line_1_2;
      AN    "HHU".Selection_Line_3_4;
      JNB   _016;
      L     '$00';
      T     "HHU".DataLine[1];
      T     "HHU".DataLine[2];
      T     "HHU".DataLine[3];
      T     "HHU".DataLine[4];
      T     "HHU".DataLine[5];
      T     "HHU".DataLine[6];
      T     "HHU".DataLine[7];
      T     "HHU".DataLine[8];
      T     "HHU".DataLine[9];
      T     "HHU".DataLine[10];
      T     "HHU".DataLine[11];
      T     "HHU".DataLine[12];
      T     "HHU".DataLine[13];
      T     "HHU".DataLine[14];
      T     "HHU".DataLine[15];
      T     "HHU".DataLine[16];
_016: NOP   0;
      A     L 15.0;
      A     "HHU".Selection_Line_1_2;
      AN    "HHU".Selection_Line_3_4;
      JNB   _017;
      L     '$00';
      T     "HHU".DataLine[1];
      T     "HHU".DataLine[2];
      T     "HHU".DataLine[3];
      T     "HHU".DataLine[4];
      T     "HHU".DataLine[5];
      L     's';
      T     "HHU".DataLine[6];
      L     'i';
      T     "HHU".DataLine[7];
      L     '$00';
      T     "HHU".DataLine[8];
      L     '2';
      T     "HHU".DataLine[9];
      L     'T';
      T     "HHU".DataLine[10];
      L     'H';
      T     "HHU".DataLine[11];
      L     '$00';
      T     "HHU".DataLine[12];
      T     "HHU".DataLine[13];
      T     "HHU".DataLine[14];
      T     "HHU".DataLine[15];
      T     "HHU".DataLine[16];
_017: NOP   0;
      A     L 15.0;
      AN    "HHU".Selection_Line_1_2;
      A     "HHU".Selection_Line_3_4;
      JNB   _018;
      L     '$00';
      T     "HHU".DataLine[1];
      T     "HHU".DataLine[2];
      T     "HHU".DataLine[3];
      T     "HHU".DataLine[4];
      T     "HHU".DataLine[5];
      L     'e';
      T     "HHU".DataLine[6];
      L     'v';
      T     "HHU".DataLine[7];
      L     'i';
      T     "HHU".DataLine[8];
      L     't';
      T     "HHU".DataLine[9];
      L     'c';
      T     "HHU".DataLine[10];
      L     'a';
      T     "HHU".DataLine[11];
      L     '$00';
      T     "HHU".DataLine[12];
      T     "HHU".DataLine[13];
      T     "HHU".DataLine[14];
      T     "HHU".DataLine[15];
      T     "HHU".DataLine[16];
_018: NOP   0;
      A     L 15.0;
      A     "HHU".Selection_Line_1_2;
      A     "HHU".Selection_Line_3_4;
      JNB   _019;
      L     '$00';
      T     "HHU".DataLine[1];
      T     "HHU".DataLine[2];
      T     "HHU".DataLine[3];
      T     "HHU".DataLine[4];
      T     "HHU".DataLine[5];
      T     "HHU".DataLine[6];
      T     "HHU".DataLine[7];
      T     "HHU".DataLine[8];
      T     "HHU".DataLine[9];
      T     "HHU".DataLine[10];
      T     "HHU".DataLine[11];
      T     "HHU".DataLine[12];
      T     "HHU".DataLine[13];
      T     "HHU".DataLine[14];
      T     "HHU".DataLine[15];
      T     "HHU".DataLine[16];
_019: NOP   0;
NETWORK
TITLE =
      AN    "HHU".Acknowledgement;
      =     "HHU".New_Data;
NETWORK
TITLE =
NETWORK
TITLE =
NETWORK
TITLE =
NETWORK
TITLE =
NETWORK
TITLE =
NETWORK
TITLE =
NETWORK
TITLE =
NETWORK
TITLE =
NETWORK
TITLE =
NETWORK
TITLE =
NETWORK
TITLE =
END_FUNCTION

FUNCTION "Share_Ctrll" : VOID	// FC 150
VERSION : 0.1
VAR_TEMP
  Ret_SFC1 : INT ;
  CDT_SFC1 : DATE_AND_TIME ;
  Ret_SFC20 : INT ;
  Ret_1 : WORD ;	//Результат работы блока FB2
  Temp1 : REAL ;
  ErrWrite : BOOL ;
  ERRCODE : INT ;
END_VAR
BEGIN
NETWORK
TITLE =
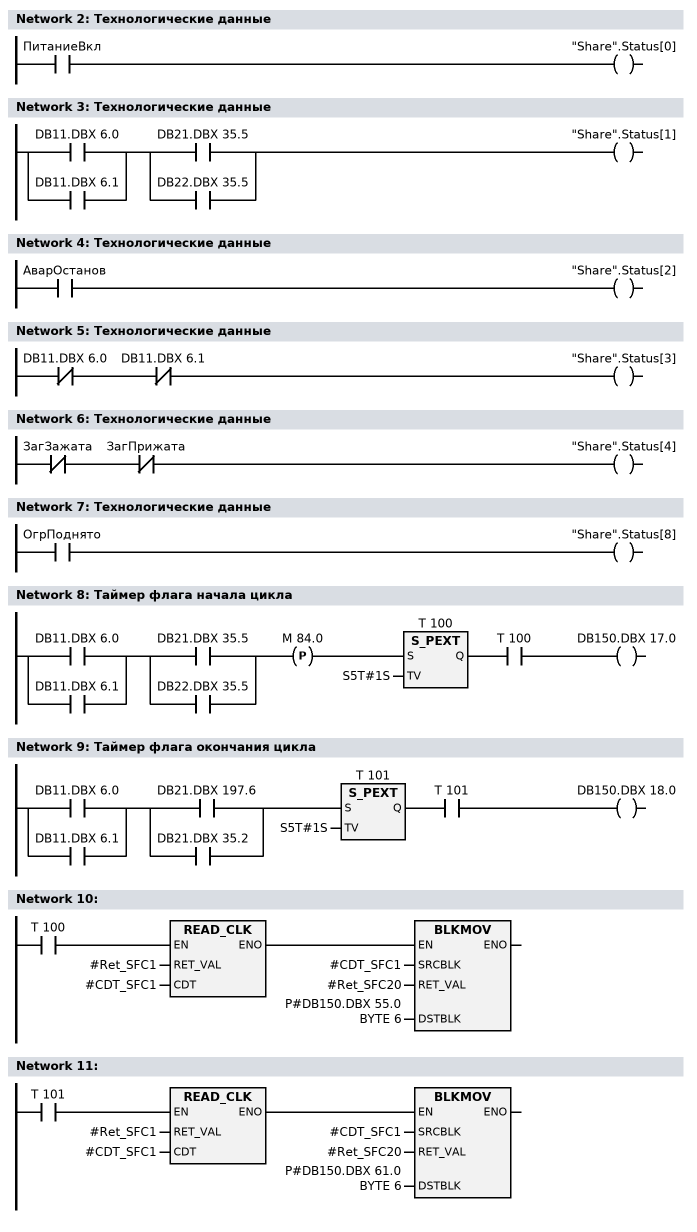
NETWORK
TITLE = Технологические данные
      A     "ПитаниеВкл";
      =     "Share".Status[0];
NETWORK
TITLE = Технологические данные
      A(;
      O     DB11.DBX 6.0;
      O     DB11.DBX 6.1;
      );
      A(;
      O     DB21.DBX 35.5;
      O     DB22.DBX 35.5;
      );
      =     "Share".Status[1];
NETWORK
TITLE = Технологические данные
//Авария.
      A     "АварОстанов";
      =     "Share".Status[2];
NETWORK
TITLE = Технологические данные
//Станок не в автомате. 
      AN    DB11.DBX 6.0;
      AN    DB11.DBX 6.1;
      =     "Share".Status[3];
NETWORK
TITLE = Технологические данные
//Заготовка не зажата.
      AN    "ЗагЗажата";
      AN    "ЗагПрижата";
      =     "Share".Status[4];
NETWORK
TITLE = Технологические данные
//Ограждение закрыто.
      A     "ОгрПоднято";
      =     "Share".Status[8];
NETWORK
TITLE = Таймер флага начала цикла
      A(;
      A(;
      O     DB11.DBX 6.0;
      O     DB11.DBX 6.1;
      );
      A(;
      O     DB21.DBX 35.5;
      O     DB22.DBX 35.5;
      );
      FP    M 84.0;
      L     S5T#1S;
      SE    T 100;
      NOP   0;
      NOP   0;
      NOP   0;
      A     T 100;
      );
      A     T 100;
      =     DB150.DBX 17.0;
NETWORK
TITLE = Таймер флага окончания цикла
      A(;
      A(;
      O     DB11.DBX 6.0;
      O     DB11.DBX 6.1;
      );
      A(;
      O     DB21.DBX 197.6;
      O     DB21.DBX 35.2;
      );
      L     S5T#1S;
      SE    T 101;
      NOP   0;
      NOP   0;
      NOP   0;
      A     T 101;
      );
      A     T 101;
      =     DB150.DBX 18.0;
NETWORK
TITLE =
      A(;
      A     T 100;
      JNB   _001;
      CALL  "READ_CLK" (
           RET_VAL                  := #Ret_SFC1,
           CDT                      := #CDT_SFC1);
_001: A     BR;
      );
      JNB   _002;
      CALL  "BLKMOV" (
           SRCBLK                   := #CDT_SFC1,
           RET_VAL                  := #Ret_SFC20,
           DSTBLK                   := P#DB150.DBX 55.0 BYTE 6);
_002: NOP   0;
NETWORK
TITLE =
      A(;
      A     T 101;
      JNB   _003;
      CALL  "READ_CLK" (
           RET_VAL                  := #Ret_SFC1,
           CDT                      := #CDT_SFC1);
_003: A     BR;
      );
      JNB   _004;
      CALL  "BLKMOV" (
           SRCBLK                   := #CDT_SFC1,
           RET_VAL                  := #Ret_SFC20,
           DSTBLK                   := P#DB150.DBX 61.0 BYTE 6);
_004: NOP   0;
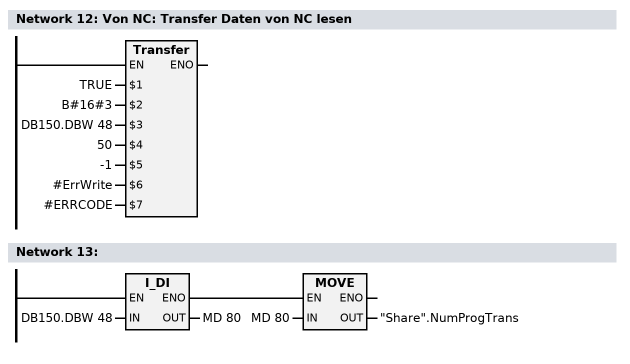
NETWORK
TITLE = Von NC: Transfer Daten von NC lesen
//$A_DBW50: Идентификатор программы обработки
      CALL  "Transfer" (
           $1                       := TRUE,
           $2                       := B#16#3,
           $3                       := DB150.DBW 48,
           $4                       := 50,
           $5                       := -1,
           $6                       := #ErrWrite,
           $7                       := #ERRCODE);
      NOP   0;
NETWORK
TITLE =
//Преобразование идентификатора программы обработки из Integer в DInteger
//
      A(;
      L     DB150.DBW 48;
      ITD;
      T     MD 80;
      SET;
      SAVE;
      CLR;
      A     BR;
      );
      JNB   _005;
      L     MD 80;
      T     "Share".NumProgTrans;
_005: NOP   0;
END_FUNCTION

// FC 1005: know-how protected block, not included

// FC 1006: know-how protected block, not included

// FC 1007: know-how protected block, not included

// FC 1008: know-how protected block, not included

// FC 1010: know-how protected block, not included

DATA_BLOCK DB 4
AUTHOR : NUMERIK
FAMILY : _800D
NAME : Basics
VERSION : 2.7
  STRUCT
   BOfeld0 : WORD  := W#16#CD54;	//Channel 1-8 ever 18 Bits
   BOfeld2 : WORD  := W#16#3553;
   BOfeld4 : WORD  := W#16#D54C;
   BOfeld6 : WORD  := W#16#5533;
   BOfeld8 : WORD  := W#16#55CD;
   BOfeld10 : WORD  := W#16#5435;
   BOfeld12 : WORD  := W#16#53D5;
   BOfeld14 : WORD  := W#16#4C55;
   BOfeld16 : WORD  := W#16#3355;
   BOfeld18 : WORD  := W#16#5555;	//18 Axes/Spindles ever 2 Bit
   BOfeld20 : WORD  := W#16#5555;
   BOfeld22 : WORD  := W#16#F5F0;	//10 User data area ever 8 Bit (Begin: DBB23)
   BOfeld24 : WORD  := W#16#F0F0;
   BOfeld26 : WORD  := W#16#F0F0;
   BOfeld28 : WORD  := W#16#F0F0;
   BOfeld30 : WORD  := W#16#F0F0;
   BOfeld32 : WORD  := W#16#F0F0;
   BOfeld34 : WORD  := W#16#F0F0;
   BOfeld36 : WORD  := W#16#F0F0;
   BOfeld38 : WORD  := W#16#F0F0;
   BOfeld40 : WORD  := W#16#F0F0;
   BOfeld42 : WORD  := W#16#F0F0;
   BOfeld44 : WORD  := W#16#F0F0;
   BOfeld46 : WORD  := W#16#F0F0;
   BOfeld48 : WORD  := W#16#F0F0;
   BOfeld50 : WORD  := W#16#F0F0;
   BOfeld52 : WORD  := W#16#F0F0;
   BOfeld54 : WORD  := W#16#F0F0;
   BOfeld56 : WORD  := W#16#F0F0;
   BOfeld58 : WORD  := W#16#F0F0;
   BOfeld60 : WORD  := W#16#F0F0;
   BOfeld62 : BYTE  := B#16#F0;
   NumUser : BYTE  := B#16#A;
   maganz : BYTE ;	//for TM, number of Magazine
   wzv : BYTE ;
   wzvdat : ARRAY  [1 .. 160 ] OF BYTE ;	//32 Magazine, possibly ever 5 Byte + Spindle
  END_STRUCT ;	
BEGIN
   BOfeld0 := W#16#CD54;
   BOfeld2 := W#16#3553;
   BOfeld4 := W#16#D54C;
   BOfeld6 := W#16#5533;
   BOfeld8 := W#16#55CD;
   BOfeld10 := W#16#5435;
   BOfeld12 := W#16#53D5;
   BOfeld14 := W#16#4C55;
   BOfeld16 := W#16#3355;
   BOfeld18 := W#16#5555;
   BOfeld20 := W#16#5555;
   BOfeld22 := W#16#F5F0;
   BOfeld24 := W#16#F0F0;
   BOfeld26 := W#16#F0F0;
   BOfeld28 := W#16#F0F0;
   BOfeld30 := W#16#F0F0;
   BOfeld32 := W#16#F0F0;
   BOfeld34 := W#16#F0F0;
   BOfeld36 := W#16#F0F0;
   BOfeld38 := W#16#F0F0;
   BOfeld40 := W#16#F0F0;
   BOfeld42 := W#16#F0F0;
   BOfeld44 := W#16#F0F0;
   BOfeld46 := W#16#F0F0;
   BOfeld48 := W#16#F0F0;
   BOfeld50 := W#16#F0F0;
   BOfeld52 := W#16#F0F0;
   BOfeld54 := W#16#F0F0;
   BOfeld56 := W#16#F0F0;
   BOfeld58 := W#16#F0F0;
   BOfeld60 := W#16#F0F0;
   BOfeld62 := B#16#F0;
   NumUser := B#16#A;
END_DATA_BLOCK

DATA_BLOCK DB 5
AUTHOR : NUMERIK
FAMILY : _800D
NAME : Basics
VERSION : 2.7
  STRUCT
   Ch1_DB2_310 : BOOL  := TRUE;	// (Channel 1-10 ever 18 Bits):  error message
   Ch1_DB2_311 : BOOL ;	// Channel 1, DB2.DBB311; operational message
   Ch1_DB2_312 : BOOL  := TRUE;	// Channel 1, DB2.DBB312; error message
   Ch1_DB2_313 : BOOL  := TRUE;	// error message
   Ch1_DB2_314 : BOOL ;	// operational message
   Ch1_DB2_315 : BOOL ;	// operational message
   Ch1_DB2_316 : BOOL  := TRUE;	// error message
   Ch1_DB2_317 : BOOL  := TRUE;	// error message
   Ch1_DB2_318 : BOOL ;	// operational message
   Ch1_DB2_319 : BOOL ;	// operational message
   Ch1_DB2_320 : BOOL  := TRUE;	// error message
   Ch1_DB2_321 : BOOL ;	// operational message
   Ch1_DB2_322 : BOOL  := TRUE;	// error message
   Ch1_DB2_323 : BOOL ;	// operational message
   Ch1_DB2_324 : BOOL  := TRUE;	// error message
   Ch1_DB2_325 : BOOL ;	// operational message
   Ch1_DB2_326 : BOOL  := TRUE;	// error message
   Ch1_DB2_327 : BOOL ;	// operational message
   Ch2_DB2_328 : BOOL  := TRUE;	// Channel 2, DB2.DBB328; error message
   Ch2_DB2_329 : BOOL ;	// Channel 2, DB2.DBB329; operational message
   Ch2_DB2_330 : BOOL  := TRUE;	// error message
   Ch2_DB2_331 : BOOL  := TRUE;	// error message
   Ch2_DB2_332 : BOOL ;	// operational message
   Ch2_DB2_333 : BOOL ;	// operational message
   Ch2_DB2_334 : BOOL  := TRUE;	// error message
   Ch2_DB2_335 : BOOL  := TRUE;	// error message
   Ch2_DB2_336 : BOOL ;	// operational message
   Ch2_DB2_337 : BOOL ;	// operational message
   Ch2_DB2_338 : BOOL  := TRUE;	// error message
   Ch2_DB2_339 : BOOL ;	// operational message
   Ch2_DB2_340 : BOOL  := TRUE;	// error message
   Ch2_DB2_341 : BOOL ;	// operational message
   Ch2_DB2_342 : BOOL  := TRUE;	// error message
   Ch2_DB2_343 : BOOL ;	// operational message
   Ch2_DB2_344 : BOOL  := TRUE;	// error message
   Ch2_DB2_345 : BOOL ;	// operational message
   Ch3_DB2_346 : BOOL  := TRUE;	// Channel 3, DB2.DBB346; error message
   Ch3_DB2_347 : BOOL ;	// Channel 3, DB2.DBB347; operational message
   Ch3_DB2_348 : BOOL  := TRUE;	// error message
   Ch3_DB2_349 : BOOL  := TRUE;	// error message
   Ch3_DB2_350 : BOOL ;	// operational message
   Ch3_DB2_351 : BOOL ;	// operational message
   Ch3_DB2_352 : BOOL  := TRUE;	// error message
   Ch3_DB2_353 : BOOL  := TRUE;	// error message
   Ch3_DB2_354 : BOOL ;	// operational message
   Ch3_DB2_355 : BOOL ;	// operational message
   Ch3_DB2_356 : BOOL  := TRUE;	// error message
   Ch3_DB2_357 : BOOL ;	// operational message
   Ch3_DB2_358 : BOOL  := TRUE;	// error message
   Ch3_DB2_359 : BOOL ;	// operational message
   Ch3_DB2_360 : BOOL  := TRUE;	// error message
   Ch3_DB2_361 : BOOL ;	// operational message
   Ch3_DB2_362 : BOOL  := TRUE;	// error message
   Ch3_DB2_363 : BOOL ;	// operational message
   Ch4_DB2_364 : BOOL  := TRUE;	// Channel 4, DB2.DBB364; error message
   Ch4_DB2_365 : BOOL ;	// Channel 4, DB2.DBB365; operational message
   Ch4_DB2_366 : BOOL  := TRUE;	// error message
   Ch4_DB2_367 : BOOL  := TRUE;	// error message
   Ch4_DB2_368 : BOOL ;	// operational message
   Ch4_DB2_369 : BOOL ;	// operational message
   Ch4_DB2_370 : BOOL  := TRUE;	// error message
   Ch4_DB2_371 : BOOL  := TRUE;	// error message
   Ch4_DB2_372 : BOOL ;	// operational message
   Ch4_DB2_373 : BOOL ;	// operational message
   Ch4_DB2_374 : BOOL  := TRUE;	// error message
   Ch4_DB2_375 : BOOL ;	// operational message
   Ch4_DB2_376 : BOOL  := TRUE;	// error message
   Ch4_DB2_377 : BOOL ;	// operational message
   Ch4_DB2_378 : BOOL  := TRUE;	// error message
   Ch4_DB2_379 : BOOL ;	// operational message
   Ch4_DB2_380 : BOOL  := TRUE;	// error message
   Ch4_DB2_381 : BOOL ;	// operational message
   Ch5_DB2_382 : BOOL  := TRUE;	// Channel 5, DB2.DBB382; error message
   Ch5_DB2_383 : BOOL ;	// Channel 5, DB2.DBB383; operational message
   Ch5_DB2_384 : BOOL  := TRUE;	// error message
   Ch5_DB2_385 : BOOL  := TRUE;	// error message
   Ch5_DB2_386 : BOOL ;	// operational message
   Ch5_DB2_387 : BOOL ;	// operational message
   Ch5_DB2_388 : BOOL  := TRUE;	// error message
   Ch5_DB2_389 : BOOL  := TRUE;	// error message
   Ch5_DB2_390 : BOOL ;	// operational message
   Ch5_DB2_391 : BOOL ;	// operational message
   Ch5_DB2_392 : BOOL  := TRUE;	// error message
   Ch5_DB2_393 : BOOL ;	// operational message
   Ch5_DB2_394 : BOOL  := TRUE;	// error message
   Ch5_DB2_395 : BOOL ;	// operational message
   Ch5_DB2_396 : BOOL  := TRUE;	// error message
   Ch5_DB2_397 : BOOL ;	// operational message
   Ch5_DB2_398 : BOOL  := TRUE;	// error message
   Ch5_DB2_399 : BOOL ;	// operational message
   Ch6_DB2_400 : BOOL  := TRUE;	// Channel 6, DB2.DBB400; error message
   Ch6_DB2_401 : BOOL ;	// Channel 6, DB2.DBB401; operational message
   Ch6_DB2_402 : BOOL  := TRUE;	// error message
   Ch6_DB2_403 : BOOL  := TRUE;	// error message
   Ch6_DB2_404 : BOOL ;	// operational message
   Ch6_DB2_405 : BOOL ;	// operational message
   Ch6_DB2_406 : BOOL  := TRUE;	// error message
   Ch6_DB2_407 : BOOL  := TRUE;	// error message
   Ch6_DB2_408 : BOOL ;	// operational message
   Ch6_DB2_409 : BOOL ;	// operational message
   Ch6_DB2_410 : BOOL  := TRUE;	// error message
   Ch6_DB2_411 : BOOL ;	// operational message
   Ch6_DB2_412 : BOOL  := TRUE;	// error message
   Ch6_DB2_413 : BOOL ;	// operational message
   Ch6_DB2_414 : BOOL  := TRUE;	// error message
   Ch6_DB2_415 : BOOL ;	// operational message
   Ch6_DB2_416 : BOOL  := TRUE;	// error message
   Ch6_DB2_417 : BOOL ;	// operational message
   Ch7_DB2_418 : BOOL  := TRUE;	// Channel 7, DB2.DBB418; error message
   Ch7_DB2_419 : BOOL ;	// Channel 7, DB2.DBB419; operational message
   Ch7_DB2_420 : BOOL  := TRUE;	// error message
   Ch7_DB2_421 : BOOL  := TRUE;	// error message
   Ch7_DB2_422 : BOOL ;	// operational message
   Ch7_DB2_423 : BOOL ;	// operational message
   Ch7_DB2_424 : BOOL  := TRUE;	// error message
   Ch7_DB2_425 : BOOL  := TRUE;	// error message
   Ch7_DB2_426 : BOOL ;	// operational message
   Ch7_DB2_427 : BOOL ;	// operational message
   Ch7_DB2_428 : BOOL  := TRUE;	// error message
   Ch7_DB2_429 : BOOL ;	// operational message
   Ch7_DB2_430 : BOOL  := TRUE;	// error message
   Ch7_DB2_431 : BOOL ;	// operational message
   Ch7_DB2_432 : BOOL  := TRUE;	// error message
   Ch7_DB2_433 : BOOL ;	// operational message
   Ch7_DB2_434 : BOOL  := TRUE;	// error message
   Ch7_DB2_435 : BOOL ;	// operational message
   Ch8_DB2_436 : BOOL  := TRUE;	// Channel 8, DB2.DBB436; error message
   Ch8_DB2_437 : BOOL ;	// Channel 8, DB2.DBB437; operational message
   Ch8_DB2_438 : BOOL  := TRUE;	// error message
   Ch8_DB2_439 : BOOL  := TRUE;	// error message
   Ch8_DB2_440 : BOOL ;	// operational message
   Ch8_DB2_441 : BOOL ;	// operational message
   Ch8_DB2_442 : BOOL  := TRUE;	// error message
   Ch8_DB2_443 : BOOL  := TRUE;	// error message
   Ch8_DB2_444 : BOOL ;	// operational message
   Ch8_DB2_445 : BOOL ;	// operational message
   Ch8_DB2_446 : BOOL  := TRUE;	// error message
   Ch8_DB2_447 : BOOL ;	// operational message
   Ch8_DB2_448 : BOOL  := TRUE;	// error message
   Ch8_DB2_449 : BOOL ;	// operational message
   Ch8_DB2_450 : BOOL  := TRUE;	// error message
   Ch8_DB2_451 : BOOL ;	// operational message
   Ch8_DB2_452 : BOOL  := TRUE;	// error message
   Ch8_DB2_453 : BOOL ;	// operational message
   Ch9_DB2_454 : BOOL  := TRUE;	// Channel 9, DB2.DBB454; error message
   Ch9_DB2_455 : BOOL ;	// Channel 9, DB2.DBB455; operational message
   Ch9_DB2_456 : BOOL  := TRUE;	// error message
   Ch9_DB2_457 : BOOL  := TRUE;	// error message
   Ch9_DB2_458 : BOOL ;	// operational message
   Ch9_DB2_459 : BOOL ;	// operational message
   Ch9_DB2_460 : BOOL  := TRUE;	// error message
   Ch9_DB2_461 : BOOL  := TRUE;	// error message
   Ch9_DB2_462 : BOOL ;	// operational message
   Ch9_DB2_463 : BOOL ;	// operational message
   Ch9_DB2_464 : BOOL  := TRUE;	// error message
   Ch9_DB2_465 : BOOL ;	// operational message
   Ch9_DB2_466 : BOOL  := TRUE;	// error message
   Ch9_DB2_467 : BOOL ;	// operational message
   Ch9_DB2_468 : BOOL  := TRUE;	// error message
   Ch9_DB2_469 : BOOL ;	// operational message
   Ch9_DB2_470 : BOOL  := TRUE;	// error message
   Ch9_DB2_471 : BOOL ;	// operational message
   Ch10_DB2_472 : BOOL  := TRUE;	// Channel 10, DB2.DBB472; error message
   Ch10_DB2_473 : BOOL ;	// Channel 10, DB2.DBB473; operational message
   Ch10_DB2_474 : BOOL  := TRUE;	// error message
   Ch10_DB2_475 : BOOL  := TRUE;	// error message
   Ch10_DB2_476 : BOOL ;	// operational message
   Ch10_DB2_477 : BOOL ;	// operational message
   Ch10_DB2_478 : BOOL  := TRUE;	// error message
   Ch10_DB2_479 : BOOL  := TRUE;	// error message
   Ch10_DB2_480 : BOOL ;	// operational message
   Ch10_DB2_481 : BOOL ;	// operational message
   Ch10_DB2_482 : BOOL  := TRUE;	// error message
   Ch10_DB2_483 : BOOL ;	// operational message
   Ch10_DB2_484 : BOOL  := TRUE;	// error message
   Ch10_DB2_485 : BOOL ;	// operational message
   Ch10_DB2_486 : BOOL  := TRUE;	// error message
   Ch10_DB2_487 : BOOL ;	// operational message
   Ch10_DB2_488 : BOOL  := TRUE;	// error message
   Ch10_DB2_489 : BOOL ;	// operational message
   Ax1_DB2_490 : BOOL  := TRUE;	// (32 Axes/Spindles ever 2 Bit):  error message
   Ax1_DB2_491 : BOOL ;	// Axis 1, DB2.DBB491; operational message
   Ax2_DB2_492 : BOOL  := TRUE;	// Axis 2, DB2.DBB492; error message
   Ax2_DB2_493 : BOOL ;	// Axis 2, DB2.DBB493; operational message
   Ax3_DB2_494 : BOOL  := TRUE;	// error message
   Ax3_DB2_495 : BOOL ;	// operational message
   Ax4_DB2_496 : BOOL  := TRUE;	// error message
   Ax4_DB2_497 : BOOL ;	// operational message
   Ax5_DB2_498 : BOOL  := TRUE;	// error message
   Ax5_DB2_499 : BOOL ;	// operational message
   Ax6_DB2_500 : BOOL  := TRUE;	// error message
   Ax6_DB2_501 : BOOL ;	// operational message
   Ax7_DB2_502 : BOOL  := TRUE;	// error message
   Ax7_DB2_503 : BOOL ;	// operational message
   Ax8_DB2_504 : BOOL  := TRUE;	// error message
   Ax8_DB2_505 : BOOL ;	// operational message
   Ax9_DB2_506 : BOOL  := TRUE;	// error message
   Ax9_DB2_507 : BOOL ;	// operational message
   Ax10_DB2_508 : BOOL  := TRUE;	// error message
   Ax10_DB2_509 : BOOL ;	// operational message
   Ax11_DB2_510 : BOOL  := TRUE;	// error message
   Ax11_DB2_511 : BOOL ;	// operational message
   Ax12_DB2_512 : BOOL  := TRUE;	// error message
   Ax12_DB2_513 : BOOL ;	// operational message
   Ax13_DB2_514 : BOOL  := TRUE;	// error message
   Ax13_DB2_515 : BOOL ;	// operational message
   Ax14_DB2_516 : BOOL  := TRUE;	// error message
   Ax14_DB2_517 : BOOL ;	// operational message
   Ax15_DB2_518 : BOOL  := TRUE;	// error message
   Ax15_DB2_519 : BOOL ;	// operational message
   Ax16_DB2_520 : BOOL  := TRUE;	// error message
   Ax16_DB2_521 : BOOL ;	// operational message
   Ax17_DB2_522 : BOOL  := TRUE;	// error message
   Ax17_DB2_523 : BOOL ;	// operational message
   Ax18_DB2_524 : BOOL  := TRUE;	// error message
   Ax18_DB2_525 : BOOL ;	// operational message
   Ax19_DB2_526 : BOOL  := TRUE;	// error message
   Ax19_DB2_527 : BOOL ;	// operational message
   Ax20_DB2_528 : BOOL  := TRUE;	// error message
   Ax20_DB2_529 : BOOL ;	// operational message
   Ax21_DB2_530 : BOOL  := TRUE;	// error message
   Ax21_DB2_531 : BOOL ;	// operational message
   Ax22_DB2_532 : BOOL  := TRUE;	// error message
   Ax22_DB2_533 : BOOL ;	// operational message
   Ax23_DB2_534 : BOOL  := TRUE;	// error message
   Ax23_DB2_535 : BOOL ;	// operational message
   Ax24_DB2_536 : BOOL  := TRUE;	// error message
   Ax24_DB2_537 : BOOL ;	// operational message
   Ax25_DB2_538 : BOOL  := TRUE;	// error message
   Ax25_DB2_539 : BOOL ;	// operational message
   Ax26_DB2_540 : BOOL  := TRUE;	// error message
   Ax26_DB2_541 : BOOL ;	// operational message
   Ax27_DB2_542 : BOOL  := TRUE;	// error message
   Ax27_DB2_543 : BOOL ;	// operational message
   Ax28_DB2_544 : BOOL  := TRUE;	// error message
   Ax28_DB2_545 : BOOL ;	// operational message
   Ax29_DB2_546 : BOOL  := TRUE;	// error message
   Ax29_DB2_547 : BOOL ;	// operational message
   Ax30_DB2_548 : BOOL  := TRUE;	// error message
   Ax30_DB2_549 : BOOL ;	// operational message
   Ax31_DB2_550 : BOOL  := TRUE;	// error message
   Ax31_DB2_551 : BOOL ;	// operational message
   Ax32_DB2_552 : BOOL  := TRUE;	// error message
   Ax32_DB2_553 : BOOL ;	// operational message
   User0_DB2_554 : BOOL  := TRUE;	// (32 User data area ever 8 Bit):  error message
   User0_DB2_555 : BOOL  := TRUE;	// UserDataArea 0, DB2.DBB555; error message
   User0_DB2_556 : BOOL  := TRUE;	// error message
   User0_DB2_557 : BOOL  := TRUE;	// error message
   User0_DB2_558 : BOOL ;	// operational message
   User0_DB2_559 : BOOL ;	// operational message
   User0_DB2_560 : BOOL ;	// operational message
   User0_DB2_561 : BOOL ;	// operational message
   User1_DB2_562 : BOOL  := TRUE;	// UserDataArea 1, DB2.DBB562; error message
   User1_DB2_563 : BOOL  := TRUE;	// error message
   User1_DB2_564 : BOOL  := TRUE;	// error message
   User1_DB2_565 : BOOL  := TRUE;	// error message
   User1_DB2_566 : BOOL ;	// operational message
   User1_DB2_567 : BOOL ;	// operational message
   User1_DB2_568 : BOOL ;	// operational message
   User1_DB2_569 : BOOL ;	// operational message
   User2_DB2_570 : BOOL  := TRUE;	// UserDataArea 2, DB2.DBB570; error message
   User2_DB2_571 : BOOL  := TRUE;	// error message
   User2_DB2_572 : BOOL  := TRUE;	// error message
   User2_DB2_573 : BOOL  := TRUE;	// error message
   User2_DB2_574 : BOOL ;	// operational message
   User2_DB2_575 : BOOL ;	// operational message
   User2_DB2_576 : BOOL ;	// operational message
   User2_DB2_577 : BOOL ;	// operational message
   User3_DB2_578 : BOOL  := TRUE;	// UserDataArea 3, DB2.DBB578; error message
   User3_DB2_579 : BOOL  := TRUE;	// error message
   User3_DB2_580 : BOOL  := TRUE;	// error message
   User3_DB2_581 : BOOL  := TRUE;	// error message
   User3_DB2_582 : BOOL ;	// operational message
   User3_DB2_583 : BOOL ;	// operational message
   User3_DB2_584 : BOOL ;	// operational message
   User3_DB2_585 : BOOL ;	// operational message
   User4_DB2_586 : BOOL  := TRUE;	// UserDataArea 4, DB2.DBB586; error message
   User4_DB2_587 : BOOL  := TRUE;	// error message
   User4_DB2_588 : BOOL  := TRUE;	// error message
   User4_DB2_589 : BOOL  := TRUE;	// error message
   User4_DB2_590 : BOOL ;	// operational message
   User4_DB2_591 : BOOL ;	// operational message
   User4_DB2_592 : BOOL ;	// operational message
   User4_DB2_593 : BOOL ;	// operational message
   User5_DB2_594 : BOOL  := TRUE;	// UserDataArea 5, DB2.DBB594; error message
   User5_DB2_595 : BOOL  := TRUE;	// error message
   User5_DB2_596 : BOOL  := TRUE;	// error message
   User5_DB2_597 : BOOL  := TRUE;	// error message
   User5_DB2_598 : BOOL ;	// operational message
   User5_DB2_599 : BOOL ;	// operational message
   User5_DB2_600 : BOOL ;	// operational message
   User5_DB2_601 : BOOL ;	// operational message
   User6_DB2_602 : BOOL  := TRUE;	// UserDataArea 6, DB2.DBB602; error message
   User6_DB2_603 : BOOL  := TRUE;	// error message
   User6_DB2_604 : BOOL  := TRUE;	// error message
   User6_DB2_605 : BOOL  := TRUE;	// error message
   User6_DB2_606 : BOOL ;	// operational message
   User6_DB2_607 : BOOL ;	// operational message
   User6_DB2_608 : BOOL ;	// operational message
   User6_DB2_609 : BOOL ;	// operational message
   User7_DB2_610 : BOOL  := TRUE;	// UserDataArea 7, DB2.DBB610; error message
   User7_DB2_611 : BOOL  := TRUE;	// error message
   User7_DB2_612 : BOOL  := TRUE;	// error message
   User7_DB2_613 : BOOL  := TRUE;	// error message
   User7_DB2_614 : BOOL ;	// operational message
   User7_DB2_615 : BOOL ;	// operational message
   User7_DB2_616 : BOOL ;	// operational message
   User7_DB2_617 : BOOL ;	// operational message
   User8_DB2_618 : BOOL  := TRUE;	// UserDataArea 8, DB2.DBB618; error message
   User8_DB2_619 : BOOL  := TRUE;	// error message
   User8_DB2_620 : BOOL  := TRUE;	// error message
   User8_DB2_621 : BOOL  := TRUE;	// error message
   User8_DB2_622 : BOOL ;	// operational message
   User8_DB2_623 : BOOL ;	// operational message
   User8_DB2_624 : BOOL ;	// operational message
   User8_DB2_625 : BOOL ;	// operational message
   User9_DB2_626 : BOOL  := TRUE;	// UserDataArea 9, DB2.DBB626; error message
   User9_DB2_627 : BOOL  := TRUE;	// error message
   User9_DB2_628 : BOOL  := TRUE;	// error message
   User9_DB2_629 : BOOL  := TRUE;	// error message
   User9_DB2_630 : BOOL ;	// operational message
   User9_DB2_631 : BOOL ;	// operational message
   User9_DB2_632 : BOOL ;	// operational message
   User9_DB2_633 : BOOL ;	// operational message
   User10_DB2_634 : BOOL  := TRUE;	// UserDataArea 10, DB2.DBB634; error message
   User10_DB2_635 : BOOL  := TRUE;	// error message
   User10_DB2_636 : BOOL  := TRUE;	// error message
   User10_DB2_637 : BOOL  := TRUE;	// error message
   User10_DB2_638 : BOOL ;	// operational message
   User10_DB2_639 : BOOL ;	// operational message
   User10_DB2_640 : BOOL ;	// operational message
   User10_DB2_641 : BOOL ;	// operational message
   User11_DB2_642 : BOOL  := TRUE;	// UserDataArea 11, DB2.DBB642; error message
   User11_DB2_643 : BOOL  := TRUE;	// error message
   User11_DB2_644 : BOOL  := TRUE;	// error message
   User11_DB2_645 : BOOL  := TRUE;	// error message
   User11_DB2_646 : BOOL ;	// operational message
   User11_DB2_647 : BOOL ;	// operational message
   User11_DB2_648 : BOOL ;	// operational message
   User11_DB2_649 : BOOL ;	// operational message
   User12_DB2_650 : BOOL  := TRUE;	// UserDataArea 12, DB2.DBB650; error message
   User12_DB2_651 : BOOL  := TRUE;	// error message
   User12_DB2_652 : BOOL  := TRUE;	// error message
   User12_DB2_653 : BOOL  := TRUE;	// error message
   User12_DB2_654 : BOOL ;	// operational message
   User12_DB2_655 : BOOL ;	// operational message
   User12_DB2_656 : BOOL ;	// operational message
   User12_DB2_657 : BOOL ;	// operational message
   User13_DB2_658 : BOOL  := TRUE;	// UserDataArea 13, DB2.DBB658; error message
   User13_DB2_659 : BOOL  := TRUE;	// error message
   User13_DB2_660 : BOOL  := TRUE;	// error message
   User13_DB2_661 : BOOL  := TRUE;	// error message
   User13_DB2_662 : BOOL ;	// operational message
   User13_DB2_663 : BOOL ;	// operational message
   User13_DB2_664 : BOOL ;	// operational message
   User13_DB2_665 : BOOL ;	// operational message
   User14_DB2_666 : BOOL  := TRUE;	// UserDataArea 14, DB2.DBB666; error message
   User14_DB2_667 : BOOL  := TRUE;	// error message
   User14_DB2_668 : BOOL  := TRUE;	// error message
   User14_DB2_669 : BOOL  := TRUE;	// error message
   User14_DB2_670 : BOOL ;	// operational message
   User14_DB2_671 : BOOL ;	// operational message
   User14_DB2_672 : BOOL ;	// operational message
   User14_DB2_673 : BOOL ;	// operational message
   User15_DB2_674 : BOOL  := TRUE;	// UserDataArea 15, DB2.DBB674; error message
   User15_DB2_675 : BOOL  := TRUE;	// error message
   User15_DB2_676 : BOOL  := TRUE;	// error message
   User15_DB2_677 : BOOL  := TRUE;	// error message
   User15_DB2_678 : BOOL ;	// operational message
   User15_DB2_679 : BOOL ;	// operational message
   User15_DB2_680 : BOOL ;	// operational message
   User15_DB2_681 : BOOL ;	// operational message
   User16_DB2_682 : BOOL  := TRUE;	// UserDataArea 16, DB2.DBB682; error message
   User16_DB2_683 : BOOL  := TRUE;	// error message
   User16_DB2_684 : BOOL  := TRUE;	// error message
   User16_DB2_685 : BOOL  := TRUE;	// error message
   User16_DB2_686 : BOOL ;	// operational message
   User16_DB2_687 : BOOL ;	// operational message
   User16_DB2_688 : BOOL ;	// operational message
   User16_DB2_689 : BOOL ;	// operational message
   User17_DB2_690 : BOOL  := TRUE;	// UserDataArea 17, DB2.DBB690; error message
   User17_DB2_691 : BOOL  := TRUE;	// error message
   User17_DB2_692 : BOOL  := TRUE;	// error message
   User17_DB2_693 : BOOL  := TRUE;	// error message
   User17_DB2_694 : BOOL ;	// operational message
   User17_DB2_695 : BOOL ;	// operational message
   User17_DB2_696 : BOOL ;	// operational message
   User17_DB2_697 : BOOL ;	// operational message
   User18_DB2_698 : BOOL  := TRUE;	// UserDataArea 18, DB2.DBB698; error message
   User18_DB2_699 : BOOL  := TRUE;	// error message
   User18_DB2_700 : BOOL  := TRUE;	// error message
   User18_DB2_701 : BOOL  := TRUE;	// error message
   User18_DB2_702 : BOOL ;	// operational message
   User18_DB2_703 : BOOL ;	// operational message
   User18_DB2_704 : BOOL ;	// operational message
   User18_DB2_705 : BOOL ;	// operational message
   User19_DB2_706 : BOOL  := TRUE;	// UserDataArea 19, DB2.DBB706; error message
   User19_DB2_707 : BOOL  := TRUE;	// error message
   User19_DB2_708 : BOOL  := TRUE;	// error message
   User19_DB2_709 : BOOL  := TRUE;	// error message
   User19_DB2_710 : BOOL ;	// operational message
   User19_DB2_711 : BOOL ;	// operational message
   User19_DB2_712 : BOOL ;	// operational message
   User19_DB2_713 : BOOL ;	// operational message
   User20_DB2_714 : BOOL  := TRUE;	// UserDataArea 20, DB2.DBB714; error message
   User20_DB2_715 : BOOL  := TRUE;	// error message
   User20_DB2_716 : BOOL  := TRUE;	// error message
   User20_DB2_717 : BOOL  := TRUE;	// error message
   User20_DB2_718 : BOOL ;	// operational message
   User20_DB2_719 : BOOL ;	// operational message
   User20_DB2_720 : BOOL ;	// operational message
   User20_DB2_721 : BOOL ;	// operational message
   User21_DB2_722 : BOOL  := TRUE;	// UserDataArea 21, DB2.DBB722; error message
   User21_DB2_723 : BOOL  := TRUE;	// error message
   User21_DB2_724 : BOOL  := TRUE;	// error message
   User21_DB2_725 : BOOL  := TRUE;	// error message
   User21_DB2_726 : BOOL ;	// operational message
   User21_DB2_727 : BOOL ;	// operational message
   User21_DB2_728 : BOOL ;	// operational message
   User21_DB2_729 : BOOL ;	// operational message
   User22_DB2_730 : BOOL  := TRUE;	// UserDataArea 22, DB2.DBB730; error message
   User22_DB2_731 : BOOL  := TRUE;	// error message
   User22_DB2_732 : BOOL  := TRUE;	// error message
   User22_DB2_733 : BOOL  := TRUE;	// error message
   User22_DB2_734 : BOOL ;	// operational message
   User22_DB2_735 : BOOL ;	// operational message
   User22_DB2_736 : BOOL ;	// operational message
   User22_DB2_737 : BOOL ;	// operational message
   User23_DB2_738 : BOOL  := TRUE;	// UserDataArea 23, DB2.DBB738; error message
   User23_DB2_739 : BOOL  := TRUE;	// error message
   User23_DB2_740 : BOOL  := TRUE;	// error message
   User23_DB2_741 : BOOL  := TRUE;	// error message
   User23_DB2_742 : BOOL ;	// operational message
   User23_DB2_743 : BOOL ;	// operational message
   User23_DB2_744 : BOOL ;	// operational message
   User23_DB2_745 : BOOL ;	// operational message
   User24_DB2_746 : BOOL  := TRUE;	// UserDataArea 24, DB2.DBB746; error message
   User24_DB2_747 : BOOL  := TRUE;	// error message
   User24_DB2_748 : BOOL  := TRUE;	// error message
   User24_DB2_749 : BOOL  := TRUE;	// error message
   User24_DB2_750 : BOOL ;	// operational message
   User24_DB2_751 : BOOL ;	// operational message
   User24_DB2_752 : BOOL ;	// operational message
   User24_DB2_753 : BOOL ;	// operational message
   User25_DB2_754 : BOOL  := TRUE;	// UserDataArea 25, DB2.DBB754; error message
   User25_DB2_755 : BOOL  := TRUE;	// error message
   User25_DB2_756 : BOOL  := TRUE;	// error message
   User25_DB2_757 : BOOL  := TRUE;	// error message
   User25_DB2_758 : BOOL ;	// operational message
   User25_DB2_759 : BOOL ;	// operational message
   User25_DB2_760 : BOOL ;	// operational message
   User25_DB2_761 : BOOL ;	// operational message
   User26_DB2_762 : BOOL  := TRUE;	// UserDataArea 26, DB2.DBB762; error message
   User26_DB2_763 : BOOL  := TRUE;	// error message
   User26_DB2_764 : BOOL  := TRUE;	// error message
   User26_DB2_765 : BOOL  := TRUE;	// error message
   User26_DB2_766 : BOOL ;	// operational message
   User26_DB2_767 : BOOL ;	// operational message
   User26_DB2_768 : BOOL ;	// operational message
   User26_DB2_769 : BOOL ;	// operational message
   User27_DB2_770 : BOOL  := TRUE;	// UserDataArea 27, DB2.DBB770; error message
   User27_DB2_771 : BOOL  := TRUE;	// error message
   User27_DB2_772 : BOOL  := TRUE;	// error message
   User27_DB2_773 : BOOL  := TRUE;	// error message
   User27_DB2_774 : BOOL ;	// operational message
   User27_DB2_775 : BOOL ;	// operational message
   User27_DB2_776 : BOOL ;	// operational message
   User27_DB2_777 : BOOL ;	// operational message
   User28_DB2_778 : BOOL  := TRUE;	// UserDataArea 28, DB2.DBB778; error message
   User28_DB2_779 : BOOL  := TRUE;	// error message
   User28_DB2_780 : BOOL  := TRUE;	// error message
   User28_DB2_781 : BOOL  := TRUE;	// error message
   User28_DB2_782 : BOOL ;	// operational message
   User28_DB2_783 : BOOL ;	// operational message
   User28_DB2_784 : BOOL ;	// operational message
   User28_DB2_785 : BOOL ;	// operational message
   User29_DB2_786 : BOOL  := TRUE;	// UserDataArea 29, DB2.DBB786; error message
   User29_DB2_787 : BOOL  := TRUE;	// error message
   User29_DB2_788 : BOOL  := TRUE;	// error message
   User29_DB2_789 : BOOL  := TRUE;	// error message
   User29_DB2_790 : BOOL ;	// operational message
   User29_DB2_791 : BOOL ;	// operational message
   User29_DB2_792 : BOOL ;	// operational message
   User29_DB2_793 : BOOL ;	// operational message
   User30_DB2_794 : BOOL  := TRUE;	// UserDataArea 30, DB2.DBB794; error message
   User30_DB2_795 : BOOL  := TRUE;	// error message
   User30_DB2_796 : BOOL  := TRUE;	// error message
   User30_DB2_797 : BOOL  := TRUE;	// error message
   User30_DB2_798 : BOOL ;	// operational message
   User30_DB2_799 : BOOL ;	// operational message
   User30_DB2_800 : BOOL ;	// operational message
   User30_DB2_801 : BOOL ;	// operational message
   User31_DB2_802 : BOOL  := TRUE;	// UserDataArea 31, DB2.DBB802; error message
   User31_DB2_803 : BOOL  := TRUE;	// error message
   User31_DB2_804 : BOOL  := TRUE;	// error message
   User31_DB2_805 : BOOL  := TRUE;	// error message
   User31_DB2_806 : BOOL ;	// operational message
   User31_DB2_807 : BOOL ;	// operational message
   User31_DB2_808 : BOOL ;	// operational message
   User31_DB2_809 : BOOL ;	// operational message
   Bit62_4 : BOOL ;	// reserved
   Bit62_5 : BOOL ;	// reserved
   Bit62_6 : BOOL ;	// reserved
   Bit62_7 : BOOL ;	// reserved
   Byte63 : BYTE ;	// reserved
   Word64 : WORD ;	// reserved
   Word66 : WORD ;	// reserved
   Word68 : WORD ;	// reserved
   Word70 : WORD ;	// reserved
   UserDek2No : ARRAY  [0 .. 31 ] OF // UserDek2No: Value 0..9 possible
   BYTE  := B#16#0;
  END_STRUCT ;	
BEGIN
   Ch1_DB2_310 := TRUE;
   Ch1_DB2_312 := TRUE;
   Ch1_DB2_313 := TRUE;
   Ch1_DB2_316 := TRUE;
   Ch1_DB2_317 := TRUE;
   Ch1_DB2_320 := TRUE;
   Ch1_DB2_322 := TRUE;
   Ch1_DB2_324 := TRUE;
   Ch1_DB2_326 := TRUE;
   Ch2_DB2_328 := TRUE;
   Ch2_DB2_330 := TRUE;
   Ch2_DB2_331 := TRUE;
   Ch2_DB2_334 := TRUE;
   Ch2_DB2_335 := TRUE;
   Ch2_DB2_338 := TRUE;
   Ch2_DB2_340 := TRUE;
   Ch2_DB2_342 := TRUE;
   Ch2_DB2_344 := TRUE;
   Ch3_DB2_346 := TRUE;
   Ch3_DB2_348 := TRUE;
   Ch3_DB2_349 := TRUE;
   Ch3_DB2_352 := TRUE;
   Ch3_DB2_353 := TRUE;
   Ch3_DB2_356 := TRUE;
   Ch3_DB2_358 := TRUE;
   Ch3_DB2_360 := TRUE;
   Ch3_DB2_362 := TRUE;
   Ch4_DB2_364 := TRUE;
   Ch4_DB2_366 := TRUE;
   Ch4_DB2_367 := TRUE;
   Ch4_DB2_370 := TRUE;
   Ch4_DB2_371 := TRUE;
   Ch4_DB2_374 := TRUE;
   Ch4_DB2_376 := TRUE;
   Ch4_DB2_378 := TRUE;
   Ch4_DB2_380 := TRUE;
   Ch5_DB2_382 := TRUE;
   Ch5_DB2_384 := TRUE;
   Ch5_DB2_385 := TRUE;
   Ch5_DB2_388 := TRUE;
   Ch5_DB2_389 := TRUE;
   Ch5_DB2_392 := TRUE;
   Ch5_DB2_394 := TRUE;
   Ch5_DB2_396 := TRUE;
   Ch5_DB2_398 := TRUE;
   Ch6_DB2_400 := TRUE;
   Ch6_DB2_402 := TRUE;
   Ch6_DB2_403 := TRUE;
   Ch6_DB2_406 := TRUE;
   Ch6_DB2_407 := TRUE;
   Ch6_DB2_410 := TRUE;
   Ch6_DB2_412 := TRUE;
   Ch6_DB2_414 := TRUE;
   Ch6_DB2_416 := TRUE;
   Ch7_DB2_418 := TRUE;
   Ch7_DB2_420 := TRUE;
   Ch7_DB2_421 := TRUE;
   Ch7_DB2_424 := TRUE;
   Ch7_DB2_425 := TRUE;
   Ch7_DB2_428 := TRUE;
   Ch7_DB2_430 := TRUE;
   Ch7_DB2_432 := TRUE;
   Ch7_DB2_434 := TRUE;
   Ch8_DB2_436 := TRUE;
   Ch8_DB2_438 := TRUE;
   Ch8_DB2_439 := TRUE;
   Ch8_DB2_442 := TRUE;
   Ch8_DB2_443 := TRUE;
   Ch8_DB2_446 := TRUE;
   Ch8_DB2_448 := TRUE;
   Ch8_DB2_450 := TRUE;
   Ch8_DB2_452 := TRUE;
   Ch9_DB2_454 := TRUE;
   Ch9_DB2_456 := TRUE;
   Ch9_DB2_457 := TRUE;
   Ch9_DB2_460 := TRUE;
   Ch9_DB2_461 := TRUE;
   Ch9_DB2_464 := TRUE;
   Ch9_DB2_466 := TRUE;
   Ch9_DB2_468 := TRUE;
   Ch9_DB2_470 := TRUE;
   Ch10_DB2_472 := TRUE;
   Ch10_DB2_474 := TRUE;
   Ch10_DB2_475 := TRUE;
   Ch10_DB2_478 := TRUE;
   Ch10_DB2_479 := TRUE;
   Ch10_DB2_482 := TRUE;
   Ch10_DB2_484 := TRUE;
   Ch10_DB2_486 := TRUE;
   Ch10_DB2_488 := TRUE;
   Ax1_DB2_490 := TRUE;
   Ax2_DB2_492 := TRUE;
   Ax3_DB2_494 := TRUE;
   Ax4_DB2_496 := TRUE;
   Ax5_DB2_498 := TRUE;
   Ax6_DB2_500 := TRUE;
   Ax7_DB2_502 := TRUE;
   Ax8_DB2_504 := TRUE;
   Ax9_DB2_506 := TRUE;
   Ax10_DB2_508 := TRUE;
   Ax11_DB2_510 := TRUE;
   Ax12_DB2_512 := TRUE;
   Ax13_DB2_514 := TRUE;
   Ax14_DB2_516 := TRUE;
   Ax15_DB2_518 := TRUE;
   Ax16_DB2_520 := TRUE;
   Ax17_DB2_522 := TRUE;
   Ax18_DB2_524 := TRUE;
   Ax19_DB2_526 := TRUE;
   Ax20_DB2_528 := TRUE;
   Ax21_DB2_530 := TRUE;
   Ax22_DB2_532 := TRUE;
   Ax23_DB2_534 := TRUE;
   Ax24_DB2_536 := TRUE;
   Ax25_DB2_538 := TRUE;
   Ax26_DB2_540 := TRUE;
   Ax27_DB2_542 := TRUE;
   Ax28_DB2_544 := TRUE;
   Ax29_DB2_546 := TRUE;
   Ax30_DB2_548 := TRUE;
   Ax31_DB2_550 := TRUE;
   Ax32_DB2_552 := TRUE;
   User0_DB2_554 := TRUE;
   User0_DB2_555 := TRUE;
   User0_DB2_556 := TRUE;
   User0_DB2_557 := TRUE;
   User1_DB2_562 := TRUE;
   User1_DB2_563 := TRUE;
   User1_DB2_564 := TRUE;
   User1_DB2_565 := TRUE;
   User2_DB2_570 := TRUE;
   User2_DB2_571 := TRUE;
   User2_DB2_572 := TRUE;
   User2_DB2_573 := TRUE;
   User3_DB2_578 := TRUE;
   User3_DB2_579 := TRUE;
   User3_DB2_580 := TRUE;
   User3_DB2_581 := TRUE;
   User4_DB2_586 := TRUE;
   User4_DB2_587 := TRUE;
   User4_DB2_588 := TRUE;
   User4_DB2_589 := TRUE;
   User5_DB2_594 := TRUE;
   User5_DB2_595 := TRUE;
   User5_DB2_596 := TRUE;
   User5_DB2_597 := TRUE;
   User6_DB2_602 := TRUE;
   User6_DB2_603 := TRUE;
   User6_DB2_604 := TRUE;
   User6_DB2_605 := TRUE;
   User7_DB2_610 := TRUE;
   User7_DB2_611 := TRUE;
   User7_DB2_612 := TRUE;
   User7_DB2_613 := TRUE;
   User8_DB2_618 := TRUE;
   User8_DB2_619 := TRUE;
   User8_DB2_620 := TRUE;
   User8_DB2_621 := TRUE;
   User9_DB2_626 := TRUE;
   User9_DB2_627 := TRUE;
   User9_DB2_628 := TRUE;
   User9_DB2_629 := TRUE;
   User10_DB2_634 := TRUE;
   User10_DB2_635 := TRUE;
   User10_DB2_636 := TRUE;
   User10_DB2_637 := TRUE;
   User11_DB2_642 := TRUE;
   User11_DB2_643 := TRUE;
   User11_DB2_644 := TRUE;
   User11_DB2_645 := TRUE;
   User12_DB2_650 := TRUE;
   User12_DB2_651 := TRUE;
   User12_DB2_652 := TRUE;
   User12_DB2_653 := TRUE;
   User13_DB2_658 := TRUE;
   User13_DB2_659 := TRUE;
   User13_DB2_660 := TRUE;
   User13_DB2_661 := TRUE;
   User14_DB2_666 := TRUE;
   User14_DB2_667 := TRUE;
   User14_DB2_668 := TRUE;
   User14_DB2_669 := TRUE;
   User15_DB2_674 := TRUE;
   User15_DB2_675 := TRUE;
   User15_DB2_676 := TRUE;
   User15_DB2_677 := TRUE;
   User16_DB2_682 := TRUE;
   User16_DB2_683 := TRUE;
   User16_DB2_684 := TRUE;
   User16_DB2_685 := TRUE;
   User17_DB2_690 := TRUE;
   User17_DB2_691 := TRUE;
   User17_DB2_692 := TRUE;
   User17_DB2_693 := TRUE;
   User18_DB2_698 := TRUE;
   User18_DB2_699 := TRUE;
   User18_DB2_700 := TRUE;
   User18_DB2_701 := TRUE;
   User19_DB2_706 := TRUE;
   User19_DB2_707 := TRUE;
   User19_DB2_708 := TRUE;
   User19_DB2_709 := TRUE;
   User20_DB2_714 := TRUE;
   User20_DB2_715 := TRUE;
   User20_DB2_716 := TRUE;
   User20_DB2_717 := TRUE;
   User21_DB2_722 := TRUE;
   User21_DB2_723 := TRUE;
   User21_DB2_724 := TRUE;
   User21_DB2_725 := TRUE;
   User22_DB2_730 := TRUE;
   User22_DB2_731 := TRUE;
   User22_DB2_732 := TRUE;
   User22_DB2_733 := TRUE;
   User23_DB2_738 := TRUE;
   User23_DB2_739 := TRUE;
   User23_DB2_740 := TRUE;
   User23_DB2_741 := TRUE;
   User24_DB2_746 := TRUE;
   User24_DB2_747 := TRUE;
   User24_DB2_748 := TRUE;
   User24_DB2_749 := TRUE;
   User25_DB2_754 := TRUE;
   User25_DB2_755 := TRUE;
   User25_DB2_756 := TRUE;
   User25_DB2_757 := TRUE;
   User26_DB2_762 := TRUE;
   User26_DB2_763 := TRUE;
   User26_DB2_764 := TRUE;
   User26_DB2_765 := TRUE;
   User27_DB2_770 := TRUE;
   User27_DB2_771 := TRUE;
   User27_DB2_772 := TRUE;
   User27_DB2_773 := TRUE;
   User28_DB2_778 := TRUE;
   User28_DB2_779 := TRUE;
   User28_DB2_780 := TRUE;
   User28_DB2_781 := TRUE;
   User29_DB2_786 := TRUE;
   User29_DB2_787 := TRUE;
   User29_DB2_788 := TRUE;
   User29_DB2_789 := TRUE;
   User30_DB2_794 := TRUE;
   User30_DB2_795 := TRUE;
   User30_DB2_796 := TRUE;
   User30_DB2_797 := TRUE;
   User31_DB2_802 := TRUE;
   User31_DB2_803 := TRUE;
   User31_DB2_804 := TRUE;
   User31_DB2_805 := TRUE;
END_DATA_BLOCK

DATA_BLOCK "gp_par"	// DB 7
TITLE = Parameters for Baseprogram
AUTHOR : NUMERIK
FAMILY : _800D
NAME : Basics
VERSION : 2.7
"RUN_UP"
BEGIN
END_DATA_BLOCK

DATA_BLOCK DB 8
AUTHOR : NUMERIK
FAMILY : _800D
NAME : Basics
VERSION : 2.7
  STRUCT
   Fc19_1 : ARRAY  [0 .. 3 ] OF BYTE ;
   Res0 : ARRAY  [0 .. 3 ] OF BYTE ;
   plData : ARRAY  [8 .. 43 ] OF BYTE ;
   TestAuto : BYTE ;
   FirstCycle : BYTE ;
   Res4 : WORD ;
   Res5 : BYTE ;
   IsFb15Correct : BYTE ;
   Res6 : ARRAY  [50 .. 61 ] OF BYTE ;
   Fc19_2 : ARRAY  [0 .. 3 ] OF BYTE ;
   Res8 : ARRAY  [66 .. 81 ] OF BYTE ;
   S7_error_id : WORD ;
   S7_error_param : WORD ;
   S7_error_adr : DWORD ;
   MinCycleTime : INT ;
   AdaptTime : INT ;
   ActCycleTime : INT ;
  END_STRUCT ;	
BEGIN
END_DATA_BLOCK

